   GP1:
	UF : 0, UT : 6,		CONFIG : 'N U T, 0, 0, 0',
	X =  -13.903  mm,	Y =   -293.878  mm,	Z =   -262.975  mm,
	W =  90.000 deg,	P =   0.000 deg,	R =   90.000 deg
};
P[961]{
   GP1:
	UF : 0, UT : 6,		CONFIG : 'N U T, 0, 0, 0',
	X =  -15.345  mm,	Y =   -294.747  mm,	Z =   -263.064  mm,
	W =  90.000 deg,	P =   0.000 deg,	R =   90.000 deg
};
P[962]{
   GP1:
	UF : 0, UT : 6,		CONFIG : 'N U T, 0, 0, 0',
	X =  -16.296  mm,	Y =   -295.198  mm,	Z =   -262.828  mm,
	W =  90.000 deg,	P =   0.000 deg,	R =   90.000 deg
};
P[963]{
   GP1:
	UF : 0, UT : 6,		CONFIG : 'N U T, 0, 0, 0',
	X =  -22.082  mm,	Y =   -298.556  mm,	Z =   -262.870  mm,
	W =  90.000 deg,	P =   0.000 deg,	R =   90.000 deg
};
P[964]{
   GP1:
	UF : 0, UT : 6,		CONFIG : 'N U T, 0, 0, 0',
	X =  -23.322  mm,	Y =   -299.338  mm,	Z =   -263.027  mm,
	W =  90.000 deg,	P =   0.000 deg,	R =   90.000 deg
};
P[965]{
   GP1:
	UF : 0, UT : 6,		CONFIG : 'N U T, 0, 0, 0',
	X =  -24.006  mm,	Y =   -299.749  mm,	Z =   -263.069  mm,
	W =  90.000 deg,	P =   0.000 deg,	R =   90.000 deg
};
P[966]{
   GP1:
	UF : 0, UT : 6,		CONFIG : 'N U T, 0, 0, 0',
	X =  -25.131  mm,	Y =   -300.448  mm,	Z =   -263.189  mm,
	W =  90.000 deg,	P =   0.000 deg,	R =   90.000 deg
};
P[967]{
   GP1:
	UF : 0, UT : 6,		CONFIG : 'N U T, 0, 0, 0',
	X =  -26.021  mm,	Y =   -300.924  mm,	Z =   -263.096  mm,
	W =  90.000 deg,	P =   0.000 deg,	R =   90.000 deg
};
P[968]{
   GP1:
	UF : 0, UT : 6,		CONFIG : 'N U T, 0, 0, 0',
	X =  -27.003  mm,	Y =   -301.481  mm,	Z =   -263.073  mm,
	W =  90.000 deg,	P =   0.000 deg,	R =   90.000 deg
};
P[969]{
   GP1:
	UF : 0, UT : 6,		CONFIG : 'N U T, 0, 0, 0',
	X =  -28.049  mm,	Y =   -302.147  mm,	Z =   -263.222  mm,
	W =  90.000 deg,	P =   0.000 deg,	R =   90.000 deg
};
P[970]{
   GP1:
	UF : 0, UT : 6,		CONFIG : 'N U T, 0, 0, 0',
	X =  -28.885  mm,	Y =   -302.634  mm,	Z =   -263.233  mm,
	W =  90.000 deg,	P =   0.000 deg,	R =   90.000 deg
};
P[971]{
   GP1:
	UF : 0, UT : 6,		CONFIG : 'N U T, 0, 0, 0',
	X =  -30.078  mm,	Y =   -303.309  mm,	Z =   -263.202  mm,
	W =  90.000 deg,	P =   0.000 deg,	R =   90.000 deg
};
P[972]{
   GP1:
	UF : 0, UT : 6,		CONFIG : 'N U T, 0, 0, 0',
	X =  -34.857  mm,	Y =   -305.939  mm,	Z =   -262.886  mm,
	W =  90.000 deg,	P =   0.000 deg,	R =   90.000 deg
};
P[973]{
   GP1:
	UF : 0, UT : 6,		CONFIG : 'N U T, 0, 0, 0',
	X =  -36.596  mm,	Y =   -307.068  mm,	Z =   -263.190  mm,
	W =  90.000 deg,	P =   0.000 deg,	R =   90.000 deg
};
P[974]{
   GP1:
	UF : 0, UT : 6,		CONFIG : 'N U T, 0, 0, 0',
	X =  -40.566  mm,	Y =   -309.197  mm,	Z =   -262.792  mm,
	W =  90.000 deg,	P =   0.000 deg,	R =   90.000 deg
};
P[975]{
   GP1:
	UF : 0, UT : 6,		CONFIG : 'N U T, 0, 0, 0',
	X =  -41.702  mm,	Y =   -309.999  mm,	Z =   -263.147  mm,
	W =  90.000 deg,	P =   0.000 deg,	R =   90.000 deg
};
P[976]{
   GP1:
	UF : 0, UT : 6,		CONFIG : 'N U T, 0, 0, 0',
	X =  -43.375  mm,	Y =   -310.890  mm,	Z =   -262.965  mm,
	W =  90.000 deg,	P =   0.000 deg,	R =   90.000 deg
};
P[977]{
   GP1:
	UF : 0, UT : 6,		CONFIG : 'N U T, 0, 0, 0',
	X =  -45.750  mm,	Y =   -312.335  mm,	Z =   -263.145  mm,
	W =  90.000 deg,	P =   0.000 deg,	R =   90.000 deg
};
P[978]{
   GP1:
	UF : 0, UT : 6,		CONFIG : 'N U T, 0, 0, 0',
	X =  -46.386  mm,	Y =   -312.642  mm,	Z =   -262.998  mm,
	W =  90.000 deg,	P =   0.000 deg,	R =   90.000 deg
};
P[979]{
   GP1:
	UF : 0, UT : 6,		CONFIG : 'N U T, 0, 0, 0',
	X =  -48.196  mm,	Y =   -313.624  mm,	Z =   -262.843  mm,
	W =  90.000 deg,	P =   0.000 deg,	R =   90.000 deg
};
P[980]{
   GP1:
	UF : 0, UT : 6,		CONFIG : 'N U T, 0, 0, 0',
	X =  -49.126  mm,	Y =   -314.230  mm,	Z =   -263.010  mm,
	W =  90.000 deg,	P =   0.000 deg,	R =   90.000 deg
};
P[981]{
   GP1:
	UF : 0, UT : 6,		CONFIG : 'N U T, 0, 0, 0',
	X =  -50.042  mm,	Y =   -314.775  mm,	Z =   -263.050  mm,
	W =  90.000 deg,	P =   0.000 deg,	R =   90.000 deg
};
P[982]{
   GP1:
	UF : 0, UT : 6,		CONFIG : 'N U T, 0, 0, 0',
	X =  -53.055  mm,	Y =   -316.565  mm,	Z =   -263.174  mm,
	W =  90.000 deg,	P =   0.000 deg,	R =   90.000 deg
};
P[983]{
   GP1:
	UF : 0, UT : 6,		CONFIG : 'N U T, 0, 0, 0',
	X =  -55.480  mm,	Y =   -317.838  mm,	Z =   -262.864  mm,
	W =  90.000 deg,	P =   0.000 deg,	R =   90.000 deg
};
P[984]{
   GP1:
	UF : 0, UT : 6,		CONFIG : 'N U T, 0, 0, 0',
	X =  -57.242  mm,	Y =   -318.967  mm,	Z =   -263.135  mm,
	W =  90.000 deg,	P =   0.000 deg,	R =   90.000 deg
};
P[985]{
   GP1:
	UF : 0, UT : 6,		CONFIG : 'N U T, 0, 0, 0',
	X =  -58.253  mm,	Y =   -319.525  mm,	Z =   -263.074  mm,
	W =  90.000 deg,	P =   0.000 deg,	R =   90.000 deg
};
P[986]{
   GP1:
	UF : 0, UT : 6,		CONFIG : 'N U T, 0, 0, 0',
	X =  -59.249  mm,	Y =   -320.111  mm,	Z =   -263.099  mm,
	W =  90.000 deg,	P =   0.000 deg,	R =   90.000 deg
};
P[987]{
   GP1:
	UF : 0, UT : 6,		CONFIG : 'N U T, 0, 0, 0',
	X =  -60.340  mm,	Y =   -320.605  mm,	Z =   -262.770  mm,
	W =  90.000 deg,	P =   0.000 deg,	R =   90.000 deg
};
P[988]{
   GP1:
	UF : 0, UT : 6,		CONFIG : 'N U T, 0, 0, 0',
	X =  -62.108  mm,	Y =   -321.686  mm,	Z =   -262.916  mm,
	W =  90.000 deg,	P =   0.000 deg,	R =   90.000 deg
};
P[989]{
   GP1:
	UF : 0, UT : 6,		CONFIG : 'N U T, 0, 0, 0',
	X =  -62.787  mm,	Y =   -322.064  mm,	Z =   -262.884  mm,
	W =  90.000 deg,	P =   0.000 deg,	R =   90.000 deg
};
P[990]{
   GP1:
	UF : 0, UT : 6,		CONFIG : 'N U T, 0, 0, 0',
	X =  -64.134  mm,	Y =   -322.855  mm,	Z =   -262.913  mm,
	W =  90.000 deg,	P =   0.000 deg,	R =   90.000 deg
};
P[991]{
   GP1:
	UF : 0, UT : 6,		CONFIG : 'N U T, 0, 0, 0',
	X =  -66.215  mm,	Y =   -324.115  mm,	Z =   -263.054  mm,
	W =  90.000 deg,	P =   0.000 deg,	R =   90.000 deg
};
P[992]{
   GP1:
	UF : 0, UT : 6,		CONFIG : 'N U T, 0, 0, 0',
	X =  -67.562  mm,	Y =   -324.948  mm,	Z =   -263.191  mm,
	W =  90.000 deg,	P =   0.000 deg,	R =   90.000 deg
};
P[993]{
   GP1:
	UF : 0, UT : 6,		CONFIG : 'N U T, 0, 0, 0',
	X =  -69.553  mm,	Y =   -326.046  mm,	Z =   -263.064  mm,
	W =  90.000 deg,	P =   0.000 deg,	R =   90.000 deg
};
P[994]{
   GP1:
	UF : 0, UT : 6,		CONFIG : 'N U T, 0, 0, 0',
	X =  -70.474  mm,	Y =   -326.519  mm,	Z =   -262.920  mm,
	W =  90.000 deg,	P =   0.000 deg,	R =   90.000 deg
};
P[995]{
   GP1:
	UF : 0, UT : 6,		CONFIG : 'N U T, 0, 0, 0',
	X =  -71.598  mm,	Y =   -327.225  mm,	Z =   -263.060  mm,
	W =  90.000 deg,	P =   0.000 deg,	R =   90.000 deg
};
P[996]{
   GP1:
	UF : 0, UT : 6,		CONFIG : 'N U T, 0, 0, 0',
	X =  -74.940  mm,	Y =   -329.214  mm,	Z =   -263.203  mm,
	W =  90.000 deg,	P =   0.000 deg,	R =   90.000 deg
};
P[997]{
   GP1:
	UF : 0, UT : 6,		CONFIG : 'N U T, 0, 0, 0',
	X =  -75.933  mm,	Y =   -329.603  mm,	Z =   -262.758  mm,
	W =  90.000 deg,	P =   0.000 deg,	R =   90.000 deg
};
P[998]{
   GP1:
	UF : 0, UT : 6,		CONFIG : 'N U T, 0, 0, 0',
	X =  -76.875  mm,	Y =   -330.326  mm,	Z =   -263.193  mm,
	W =  90.000 deg,	P =   0.000 deg,	R =   90.000 deg
};
P[999]{
   GP1:
	UF : 0, UT : 6,		CONFIG : 'N U T, 0, 0, 0',
	X =  -79.257  mm,	Y =   -331.581  mm,	Z =   -262.899  mm,
	W =  90.000 deg,	P =   0.000 deg,	R =   90.000 deg
};
P[1000]{
   GP1:
	UF : 0, UT : 6,		CONFIG : 'N U T, 0, 0, 0',
	X =  -80.224  mm,	Y =   -332.210  mm,	Z =   -263.072  mm,
	W =  90.000 deg,	P =   0.000 deg,	R =   90.000 deg
};
P[1001]{
   GP1:
	UF : 0, UT : 6,		CONFIG : 'N U T, 0, 0, 0',
	X =  -81.301  mm,	Y =   -332.796  mm,	Z =   -262.984  mm,
	W =  90.000 deg,	P =   0.000 deg,	R =   90.000 deg
};
P[1002]{
   GP1:
	UF : 0, UT : 6,		CONFIG : 'N U T, 0, 0, 0',
	X =  -82.537  mm,	Y =   -333.595  mm,	Z =   -263.191  mm,
	W =  90.000 deg,	P =   0.000 deg,	R =   90.000 deg
};
P[1003]{
   GP1:
	UF : 0, UT : 6,		CONFIG : 'N U T, 0, 0, 0',
	X =  -84.221  mm,	Y =   -334.495  mm,	Z =   -263.013  mm,
	W =  90.000 deg,	P =   0.000 deg,	R =   90.000 deg
};
P[1004]{
   GP1:
	UF : 0, UT : 6,		CONFIG : 'N U T, 0, 0, 0',
	X =  -86.503  mm,	Y =   -335.901  mm,	Z =   -263.231  mm,
	W =  90.000 deg,	P =   0.000 deg,	R =   90.000 deg
};
P[1005]{
   GP1:
	UF : 0, UT : 6,		CONFIG : 'N U T, 0, 0, 0',
	X =  -87.830  mm,	Y =   -336.582  mm,	Z =   -263.024  mm,
	W =  90.000 deg,	P =   0.000 deg,	R =   90.000 deg
};
P[1006]{
   GP1:
	UF : 0, UT : 6,		CONFIG : 'N U T, 0, 0, 0',
	X =  -88.563  mm,	Y =   -336.971  mm,	Z =   -262.940  mm,
	W =  90.000 deg,	P =   0.000 deg,	R =   90.000 deg
};
P[1007]{
   GP1:
	UF : 0, UT : 6,		CONFIG : 'N U T, 0, 0, 0',
	X =  -91.169  mm,	Y =   -338.484  mm,	Z =   -262.960  mm,
	W =  90.000 deg,	P =   0.000 deg,	R =   90.000 deg
};
P[1008]{
   GP1:
	UF : 0, UT : 6,		CONFIG : 'N U T, 0, 0, 0',
	X =  -91.807  mm,	Y =   -338.966  mm,	Z =   -263.237  mm,
	W =  90.000 deg,	P =   0.000 deg,	R =   90.000 deg
};
P[1009]{
   GP1:
	UF : 0, UT : 6,		CONFIG : 'N U T, 0, 0, 0',
	X =  -92.493  mm,	Y =   -339.305  mm,	Z =   -263.100  mm,
	W =  90.000 deg,	P =   0.000 deg,	R =   90.000 deg
};
P[1010]{
   GP1:
	UF : 0, UT : 6,		CONFIG : 'N U T, 0, 0, 0',
	X =  -93.733  mm,	Y =   -340.067  mm,	Z =   -263.210  mm,
	W =  90.000 deg,	P =   0.000 deg,	R =   90.000 deg
};
P[1011]{
   GP1:
	UF : 0, UT : 6,		CONFIG : 'N U T, 0, 0, 0',
	X =  -95.528  mm,	Y =   -341.015  mm,	Z =   -262.997  mm,
	W =  90.000 deg,	P =   0.000 deg,	R =   90.000 deg
};
P[1012]{
   GP1:
	UF : 0, UT : 6,		CONFIG : 'N U T, 0, 0, 0',
	X =  -96.099  mm,	Y =   -341.423  mm,	Z =   -263.185  mm,
	W =  90.000 deg,	P =   0.000 deg,	R =   90.000 deg
};
P[1013]{
   GP1:
	UF : 0, UT : 6,		CONFIG : 'N U T, 0, 0, 0',
	X =  -97.870  mm,	Y =   -342.351  mm,	Z =   -262.957  mm,
	W =  90.000 deg,	P =   0.000 deg,	R =   90.000 deg
};
P[1014]{
   GP1:
	UF : 0, UT : 6,		CONFIG : 'N U T, 0, 0, 0',
	X =  -98.558  mm,	Y =   -342.684  mm,	Z =   -262.799  mm,
	W =  90.000 deg,	P =   0.000 deg,	R =   90.000 deg
};
P[1015]{
   GP1:
	UF : 0, UT : 6,		CONFIG : 'N U T, 0, 0, 0',
	X =  -100.265  mm,	Y =   -343.664  mm,	Z =   -262.786  mm,
	W =  90.000 deg,	P =   0.000 deg,	R =   90.000 deg
};
P[1016]{
   GP1:
	UF : 0, UT : 6,		CONFIG : 'N U T, 0, 0, 0',
	X =  -101.104  mm,	Y =   -344.315  mm,	Z =   -263.189  mm,
	W =  90.000 deg,	P =   0.000 deg,	R =   90.000 deg
};
P[1017]{
   GP1:
	UF : 0, UT : 6,		CONFIG : 'N U T, 0, 0, 0',
	X =  -102.677  mm,	Y =   -345.092  mm,	Z =   -262.871  mm,
	W =  90.000 deg,	P =   0.000 deg,	R =   90.000 deg
};
P[1018]{
   GP1:
	UF : 0, UT : 6,		CONFIG : 'N U T, 0, 0, 0',
	X =  -103.616  mm,	Y =   -345.734  mm,	Z =   -263.113  mm,
	W =  90.000 deg,	P =   0.000 deg,	R =   90.000 deg
};
P[1019]{
   GP1:
	UF : 0, UT : 6,		CONFIG : 'N U T, 0, 0, 0',
	X =  -107.113  mm,	Y =   -347.775  mm,	Z =   -263.168  mm,
	W =  90.000 deg,	P =   0.000 deg,	R =   90.000 deg
};
P[1020]{
   GP1:
	UF : 0, UT : 6,		CONFIG : 'N U T, 0, 0, 0',
	X =  -109.559  mm,	Y =   -349.127  mm,	Z =   -263.019  mm,
	W =  90.000 deg,	P =   0.000 deg,	R =   90.000 deg
};
P[1021]{
   GP1:
	UF : 0, UT : 6,		CONFIG : 'N U T, 0, 0, 0',
	X =  -110.422  mm,	Y =   -349.715  mm,	Z =   -263.238  mm,
	W =  90.000 deg,	P =   0.000 deg,	R =   90.000 deg
};
P[1022]{
   GP1:
	UF : 0, UT : 6,		CONFIG : 'N U T, 0, 0, 0',
	X =  -111.709  mm,	Y =   -350.433  mm,	Z =   -263.142  mm,
	W =  90.000 deg,	P =   0.000 deg,	R =   90.000 deg
};
P[1023]{
   GP1:
	UF : 0, UT : 6,		CONFIG : 'N U T, 0, 0, 0',
	X =  -114.563  mm,	Y =   -352.669  mm,	Z =   -263.167  mm,
	W =  90.000 deg,	P =   0.000 deg,	R =   90.000 deg
};
P[1024]{
   GP1:
	UF : 0, UT : 6,		CONFIG : 'N U T, 0, 0, 0',
	X =  -115.198  mm,	Y =   -353.316  mm,	Z =   -263.069  mm,
	W =  90.000 deg,	P =   0.000 deg,	R =   90.000 deg
};
P[1025]{
   GP1:
	UF : 0, UT : 6,		CONFIG : 'N U T, 0, 0, 0',
	X =  -117.423  mm,	Y =   -356.705  mm,	Z =   -263.118  mm,
	W =  90.000 deg,	P =   0.000 deg,	R =   90.000 deg
};
P[1026]{
   GP1:
	UF : 0, UT : 6,		CONFIG : 'N U T, 0, 0, 0',
	X =  -117.726  mm,	Y =   -357.586  mm,	Z =   -263.245  mm,
	W =  90.000 deg,	P =   0.000 deg,	R =   90.000 deg
};
P[1027]{
   GP1:
	UF : 0, UT : 6,		CONFIG : 'N U T, 0, 0, 0',
	X =  -118.115  mm,	Y =   -358.723  mm,	Z =   -263.116  mm,
	W =  90.000 deg,	P =   0.000 deg,	R =   90.000 deg
};
P[1028]{
   GP1:
	UF : 0, UT : 6,		CONFIG : 'N U T, 0, 0, 0',
	X =  -118.602  mm,	Y =   -361.256  mm,	Z =   -262.992  mm,
	W =  90.000 deg,	P =   0.000 deg,	R =   90.000 deg
};
P[1029]{
   GP1:
	UF : 0, UT : 6,		CONFIG : 'N U T, 0, 0, 0',
	X =  -118.574  mm,	Y =   -363.321  mm,	Z =   -263.077  mm,
	W =  90.000 deg,	P =   0.000 deg,	R =   90.000 deg
};
P[1030]{
   GP1:
	UF : 0, UT : 6,		CONFIG : 'N U T, 0, 0, 0',
	X =  -118.207  mm,	Y =   -365.061  mm,	Z =   -263.179  mm,
	W =  90.000 deg,	P =   0.000 deg,	R =   90.000 deg
};
P[1031]{
   GP1:
	UF : 0, UT : 6,		CONFIG : 'N U T, 0, 0, 0',
	X =  -117.889  mm,	Y =   -366.383  mm,	Z =   -263.224  mm,
	W =  90.000 deg,	P =   0.000 deg,	R =   90.000 deg
};
P[1032]{
   GP1:
	UF : 0, UT : 6,		CONFIG : 'N U T, 0, 0, 0',
	X =  -117.012  mm,	Y =   -368.554  mm,	Z =   -263.053  mm,
	W =  90.000 deg,	P =   0.000 deg,	R =   90.000 deg
};
P[1033]{
   GP1:
	UF : 0, UT : 6,		CONFIG : 'N U T, 0, 0, 0',
	X =  -116.322  mm,	Y =   -369.824  mm,	Z =   -263.139  mm,
	W =  90.000 deg,	P =   0.000 deg,	R =   90.000 deg
};
P[1034]{
   GP1:
	UF : 0, UT : 6,		CONFIG : 'N U T, 0, 0, 0',
	X =  -115.983  mm,	Y =   -370.432  mm,	Z =   -263.111  mm,
	W =  90.000 deg,	P =   0.000 deg,	R =   90.000 deg
};
P[1035]{
   GP1:
	UF : 0, UT : 6,		CONFIG : 'N U T, 0, 0, 0',
	X =  -115.285  mm,	Y =   -371.743  mm,	Z =   -262.966  mm,
	W =  90.000 deg,	P =   0.000 deg,	R =   90.000 deg
};
P[1036]{
   GP1:
	UF : 0, UT : 6,		CONFIG : 'N U T, 0, 0, 0',
	X =  -114.882  mm,	Y =   -372.354  mm,	Z =   -263.089  mm,
	W =  90.000 deg,	P =   0.000 deg,	R =   90.000 deg
};
P[1037]{
   GP1:
	UF : 0, UT : 6,		CONFIG : 'N U T, 0, 0, 0',
	X =  -113.584  mm,	Y =   -374.650  mm,	Z =   -263.021  mm,
	W =  90.000 deg,	P =   0.000 deg,	R =   90.000 deg
};
P[1038]{
   GP1:
	UF : 0, UT : 6,		CONFIG : 'N U T, 0, 0, 0',
	X =  -112.392  mm,	Y =   -376.883  mm,	Z =   -262.787  mm,
	W =  90.000 deg,	P =   0.000 deg,	R =   90.000 deg
};
P[1039]{
   GP1:
	UF : 0, UT : 6,		CONFIG : 'N U T, 0, 0, 0',
	X =  -111.637  mm,	Y =   -377.966  mm,	Z =   -263.099  mm,
	W =  90.000 deg,	P =   0.000 deg,	R =   90.000 deg
};
P[1040]{
   GP1:
	UF : 0, UT : 6,		CONFIG : 'N U T, 0, 0, 0',
	X =  -107.435  mm,	Y =   -385.253  mm,	Z =   -263.085  mm,
	W =  90.000 deg,	P =   0.000 deg,	R =   90.000 deg
};
P[1041]{
   GP1:
	UF : 0, UT : 6,		CONFIG : 'N U T, 0, 0, 0',
	X =  -106.804  mm,	Y =   -386.568  mm,	Z =   -262.775  mm,
	W =  90.000 deg,	P =   0.000 deg,	R =   90.000 deg
};
P[1042]{
   GP1:
	UF : 0, UT : 6,		CONFIG : 'N U T, 0, 0, 0',
	X =  -105.774  mm,	Y =   -388.206  mm,	Z =   -262.982  mm,
	W =  90.000 deg,	P =   0.000 deg,	R =   90.000 deg
};
P[1043]{
   GP1:
	UF : 0, UT : 6,		CONFIG : 'N U T, 0, 0, 0',
	X =  -105.097  mm,	Y =   -389.195  mm,	Z =   -263.237  mm,
	W =  90.000 deg,	P =   0.000 deg,	R =   90.000 deg
};
P[1044]{
   GP1:
	UF : 0, UT : 6,		CONFIG : 'N U T, 0, 0, 0',
	X =  -104.414  mm,	Y =   -390.491  mm,	Z =   -263.078  mm,
	W =  90.000 deg,	P =   0.000 deg,	R =   90.000 deg
};
P[1045]{
   GP1:
	UF : 0, UT : 6,		CONFIG : 'N U T, 0, 0, 0',
	X =  -103.894  mm,	Y =   -391.411  mm,	Z =   -263.052  mm,
	W =  90.000 deg,	P =   0.000 deg,	R =   90.000 deg
};
P[1046]{
   GP1:
	UF : 0, UT : 6,		CONFIG : 'N U T, 0, 0, 0',
	X =  -103.256  mm,	Y =   -392.421  mm,	Z =   -263.184  mm,
	W =  90.000 deg,	P =   0.000 deg,	R =   90.000 deg
};
P[1047]{
   GP1:
	UF : 0, UT : 6,		CONFIG : 'N U T, 0, 0, 0',
	X =  -102.760  mm,	Y =   -393.344  mm,	Z =   -263.095  mm,
	W =  90.000 deg,	P =   0.000 deg,	R =   90.000 deg
};
P[1048]{
   GP1:
	UF : 0, UT : 6,		CONFIG : 'N U T, 0, 0, 0',
	X =  -101.499  mm,	Y =   -395.746  mm,	Z =   -262.790  mm,
	W =  90.000 deg,	P =   0.000 deg,	R =   90.000 deg
};
P[1049]{
   GP1:
	UF : 0, UT : 6,		CONFIG : 'N U T, 0, 0, 0',
	X =  -100.798  mm,	Y =   -396.817  mm,	Z =   -262.989  mm,
	W =  90.000 deg,	P =   0.000 deg,	R =   90.000 deg
};
P[1050]{
   GP1:
	UF : 0, UT : 6,		CONFIG : 'N U T, 0, 0, 0',
	X =  -99.795  mm,	Y =   -398.512  mm,	Z =   -263.050  mm,
	W =  90.000 deg,	P =   0.000 deg,	R =   90.000 deg
};
P[1051]{
   GP1:
	UF : 0, UT : 6,		CONFIG : 'N U T, 0, 0, 0',
	X =  -99.179  mm,	Y =   -399.555  mm,	Z =   -263.082  mm,
	W =  90.000 deg,	P =   0.000 deg,	R =   90.000 deg
};
P[1052]{
   GP1:
	UF : 0, UT : 6,		CONFIG : 'N U T, 0, 0, 0',
	X =  -97.942  mm,	Y =   -401.662  mm,	Z =   -263.134  mm,
	W =  90.000 deg,	P =   0.000 deg,	R =   90.000 deg
};
P[1053]{
   GP1:
	UF : 0, UT : 6,		CONFIG : 'N U T, 0, 0, 0',
	X =  -97.334  mm,	Y =   -402.964  mm,	Z =   -262.783  mm,
	W =  90.000 deg,	P =   0.000 deg,	R =   90.000 deg
};
P[1054]{
   GP1:
	UF : 0, UT : 6,		CONFIG : 'N U T, 0, 0, 0',
	X =  -96.595  mm,	Y =   -404.228  mm,	Z =   -262.806  mm,
	W =  90.000 deg,	P =   0.000 deg,	R =   90.000 deg
};
P[1055]{
   GP1:
	UF : 0, UT : 6,		CONFIG : 'N U T, 0, 0, 0',
	X =  -95.365  mm,	Y =   -406.151  mm,	Z =   -263.096  mm,
	W =  90.000 deg,	P =   0.000 deg,	R =   90.000 deg
};
P[1056]{
   GP1:
	UF : 0, UT : 6,		CONFIG : 'N U T, 0, 0, 0',
	X =  -94.824  mm,	Y =   -407.301  mm,	Z =   -262.797  mm,
	W =  90.000 deg,	P =   0.000 deg,	R =   90.000 deg
};
P[1057]{
   GP1:
	UF : 0, UT : 6,		CONFIG : 'N U T, 0, 0, 0',
	X =  -93.955  mm,	Y =   -408.499  mm,	Z =   -263.227  mm,
	W =  90.000 deg,	P =   0.000 deg,	R =   90.000 deg
};
P[1058]{
   GP1:
	UF : 0, UT : 6,		CONFIG : 'N U T, 0, 0, 0',
	X =  -93.580  mm,	Y =   -409.387  mm,	Z =   -262.895  mm,
	W =  90.000 deg,	P =   0.000 deg,	R =   90.000 deg
};
P[1059]{
   GP1:
	UF : 0, UT : 6,		CONFIG : 'N U T, 0, 0, 0',
	X =  -92.695  mm,	Y =   -410.733  mm,	Z =   -263.155  mm,
	W =  90.000 deg,	P =   0.000 deg,	R =   90.000 deg
};
P[1060]{
   GP1:
	UF : 0, UT : 6,		CONFIG : 'N U T, 0, 0, 0',
	X =  -90.502  mm,	Y =   -414.497  mm,	Z =   -263.203  mm,
	W =  90.000 deg,	P =   0.000 deg,	R =   90.000 deg
};
P[1061]{
   GP1:
	UF : 0, UT : 6,		CONFIG : 'N U T, 0, 0, 0',
	X =  -89.845  mm,	Y =   -415.741  mm,	Z =   -263.054  mm,
	W =  90.000 deg,	P =   0.000 deg,	R =   90.000 deg
};
P[1062]{
   GP1:
	UF : 0, UT : 6,		CONFIG : 'N U T, 0, 0, 0',
	X =  -89.462  mm,	Y =   -416.470  mm,	Z =   -262.962  mm,
	W =  90.000 deg,	P =   0.000 deg,	R =   90.000 deg
};
P[1063]{
   GP1:
	UF : 0, UT : 6,		CONFIG : 'N U T, 0, 0, 0',
	X =  -89.089  mm,	Y =   -417.185  mm,	Z =   -262.868  mm,
	W =  90.000 deg,	P =   0.000 deg,	R =   90.000 deg
};
P[1064]{
   GP1:
	UF : 0, UT : 6,		CONFIG : 'N U T, 0, 0, 0',
	X =  -87.684  mm,	Y =   -419.644  mm,	Z =   -262.831  mm,
	W =  90.000 deg,	P =   0.000 deg,	R =   90.000 deg
};
P[1065]{
   GP1:
	UF : 0, UT : 6,		CONFIG : 'N U T, 0, 0, 0',
	X =  -87.091  mm,	Y =   -420.612  mm,	Z =   -262.912  mm,
	W =  90.000 deg,	P =   0.000 deg,	R =   90.000 deg
};
P[1066]{
   GP1:
	UF : 0, UT : 6,		CONFIG : 'N U T, 0, 0, 0',
	X =  -86.461  mm,	Y =   -421.515  mm,	Z =   -263.175  mm,
	W =  90.000 deg,	P =   0.000 deg,	R =   90.000 deg
};
P[1067]{
   GP1:
	UF : 0, UT : 6,		CONFIG : 'N U T, 0, 0, 0',
	X =  -85.753  mm,	Y =   -422.744  mm,	Z =   -263.173  mm,
	W =  90.000 deg,	P =   0.000 deg,	R =   90.000 deg
};
P[1068]{
   GP1:
	UF : 0, UT : 6,		CONFIG : 'N U T, 0, 0, 0',
	X =  -84.853  mm,	Y =   -424.493  mm,	Z =   -262.904  mm,
	W =  90.000 deg,	P =   0.000 deg,	R =   90.000 deg
};
P[1069]{
   GP1:
	UF : 0, UT : 6,		CONFIG : 'N U T, 0, 0, 0',
	X =  -82.147  mm,	Y =   -428.978  mm,	Z =   -263.189  mm,
	W =  90.000 deg,	P =   0.000 deg,	R =   90.000 deg
};
P[1070]{
   GP1:
	UF : 0, UT : 6,		CONFIG : 'N U T, 0, 0, 0',
	X =  -81.488  mm,	Y =   -430.368  mm,	Z =   -262.838  mm,
	W =  90.000 deg,	P =   0.000 deg,	R =   90.000 deg
};
P[1071]{
   GP1:
	UF : 0, UT : 6,		CONFIG : 'N U T, 0, 0, 0',
	X =  -80.821  mm,	Y =   -431.485  mm,	Z =   -262.895  mm,
	W =  90.000 deg,	P =   0.000 deg,	R =   90.000 deg
};
P[1072]{
   GP1:
	UF : 0, UT : 6,		CONFIG : 'N U T, 0, 0, 0',
	X =  -80.262  mm,	Y =   -432.225  mm,	Z =   -263.213  mm,
	W =  90.000 deg,	P =   0.000 deg,	R =   90.000 deg
};
P[1073]{
   GP1:
	UF : 0, UT : 6,		CONFIG : 'N U T, 0, 0, 0',
	X =  -78.623  mm,	Y =   -435.273  mm,	Z =   -262.917  mm,
	W =  90.000 deg,	P =   0.000 deg,	R =   90.000 deg
};
P[1074]{
   GP1:
	UF : 0, UT : 6,		CONFIG : 'N U T, 0, 0, 0',
	X =  -77.822  mm,	Y =   -436.615  mm,	Z =   -262.983  mm,
	W =  90.000 deg,	P =   0.000 deg,	R =   90.000 deg
};
P[1075]{
   GP1:
	UF : 0, UT : 6,		CONFIG : 'N U T, 0, 0, 0',
	X =  -77.155  mm,	Y =   -437.636  mm,	Z =   -263.172  mm,
	W =  90.000 deg,	P =   0.000 deg,	R =   90.000 deg
};
P[1076]{
   GP1:
	UF : 0, UT : 6,		CONFIG : 'N U T, 0, 0, 0',
	X =  -76.150  mm,	Y =   -439.438  mm,	Z =   -263.086  mm,
	W =  90.000 deg,	P =   0.000 deg,	R =   90.000 deg
};
P[1077]{
   GP1:
	UF : 0, UT : 6,		CONFIG : 'N U T, 0, 0, 0',
	X =  -75.497  mm,	Y =   -440.686  mm,	Z =   -262.922  mm,
	W =  90.000 deg,	P =   0.000 deg,	R =   90.000 deg
};
P[1078]{
   GP1:
	UF : 0, UT : 6,		CONFIG : 'N U T, 0, 0, 0',
	X =  -73.747  mm,	Y =   -443.722  mm,	Z =   -262.912  mm,
	W =  90.000 deg,	P =   0.000 deg,	R =   90.000 deg
};
P[1079]{
   GP1:
	UF : 0, UT : 6,		CONFIG : 'N U T, 0, 0, 0',
	X =  -73.249  mm,	Y =   -444.554  mm,	Z =   -262.957  mm,
	W =  90.000 deg,	P =   0.000 deg,	R =   90.000 deg
};
P[1080]{
   GP1:
	UF : 0, UT : 6,		CONFIG : 'N U T, 0, 0, 0',
	X =  -72.020  mm,	Y =   -446.678  mm,	Z =   -262.963  mm,
	W =  90.000 deg,	P =   0.000 deg,	R =   90.000 deg
};
P[1081]{
   GP1:
	UF : 0, UT : 6,		CONFIG : 'N U T, 0, 0, 0',
	X =  -71.491  mm,	Y =   -447.557  mm,	Z =   -263.017  mm,
	W =  90.000 deg,	P =   0.000 deg,	R =   90.000 deg
};
P[1082]{
   GP1:
	UF : 0, UT : 6,		CONFIG : 'N U T, 0, 0, 0',
	X =  -68.260  mm,	Y =   -453.237  mm,	Z =   -262.897  mm,
	W =  90.000 deg,	P =   0.000 deg,	R =   90.000 deg
};
P[1083]{
   GP1:
	UF : 0, UT : 6,		CONFIG : 'N U T, 0, 0, 0',
	X =  -66.554  mm,	Y =   -456.053  mm,	Z =   -263.092  mm,
	W =  90.000 deg,	P =   0.000 deg,	R =   90.000 deg
};
P[1084]{
   GP1:
	UF : 0, UT : 6,		CONFIG : 'N U T, 0, 0, 0',
	X =  -64.066  mm,	Y =   -460.264  mm,	Z =   -263.227  mm,
	W =  90.000 deg,	P =   0.000 deg,	R =   90.000 deg
};
P[1085]{
   GP1:
	UF : 0, UT : 6,		CONFIG : 'N U T, 0, 0, 0',
	X =  -63.745  mm,	Y =   -461.131  mm,	Z =   -262.793  mm,
	W =  90.000 deg,	P =   0.000 deg,	R =   90.000 deg
};
P[1086]{
   GP1:
	UF : 0, UT : 6,		CONFIG : 'N U T, 0, 0, 0',
	X =  -61.359  mm,	Y =   -464.951  mm,	Z =   -263.231  mm,
	W =  90.000 deg,	P =   0.000 deg,	R =   90.000 deg
};
P[1087]{
   GP1:
	UF : 0, UT : 6,		CONFIG : 'N U T, 0, 0, 0',
	X =  -60.085  mm,	Y =   -467.217  mm,	Z =   -263.147  mm,
	W =  90.000 deg,	P =   0.000 deg,	R =   90.000 deg
};
P[1088]{
   GP1:
	UF : 0, UT : 6,		CONFIG : 'N U T, 0, 0, 0',
	X =  -59.296  mm,	Y =   -468.735  mm,	Z =   -262.934  mm,
	W =  90.000 deg,	P =   0.000 deg,	R =   90.000 deg
};
P[1089]{
   GP1:
	UF : 0, UT : 6,		CONFIG : 'N U T, 0, 0, 0',
	X =  -58.716  mm,	Y =   -469.717  mm,	Z =   -262.965  mm,
	W =  90.000 deg,	P =   0.000 deg,	R =   90.000 deg
};
P[1090]{
   GP1:
	UF : 0, UT : 6,		CONFIG : 'N U T, 0, 0, 0',
	X =  -58.101  mm,	Y =   -470.743  mm,	Z =   -263.019  mm,
	W =  90.000 deg,	P =   0.000 deg,	R =   90.000 deg
};
P[1091]{
   GP1:
	UF : 0, UT : 6,		CONFIG : 'N U T, 0, 0, 0',
	X =  -57.668  mm,	Y =   -471.616  mm,	Z =   -262.847  mm,
	W =  90.000 deg,	P =   0.000 deg,	R =   90.000 deg
};
P[1092]{
   GP1:
	UF : 0, UT : 6,		CONFIG : 'N U T, 0, 0, 0',
	X =  -56.102  mm,	Y =   -474.080  mm,	Z =   -263.194  mm,
	W =  90.000 deg,	P =   0.000 deg,	R =   90.000 deg
};
P[1093]{
   GP1:
	UF : 0, UT : 6,		CONFIG : 'N U T, 0, 0, 0',
	X =  -54.772  mm,	Y =   -476.607  mm,	Z =   -262.882  mm,
	W =  90.000 deg,	P =   0.000 deg,	R =   90.000 deg
};
P[1094]{
   GP1:
	UF : 0, UT : 6,		CONFIG : 'N U T, 0, 0, 0',
	X =  -53.834  mm,	Y =   -478.104  mm,	Z =   -263.060  mm,
	W =  90.000 deg,	P =   0.000 deg,	R =   90.000 deg
};
P[1095]{
   GP1:
	UF : 0, UT : 6,		CONFIG : 'N U T, 0, 0, 0',
	X =  -53.421  mm,	Y =   -478.798  mm,	Z =   -263.091  mm,
	W =  90.000 deg,	P =   0.000 deg,	R =   90.000 deg
};
P[1096]{
   GP1:
	UF : 0, UT : 6,		CONFIG : 'N U T, 0, 0, 0',
	X =  -52.867  mm,	Y =   -479.903  mm,	Z =   -262.889  mm,
	W =  90.000 deg,	P =   0.000 deg,	R =   90.000 deg
};
P[1097]{
   GP1:
	UF : 0, UT : 6,		CONFIG : 'N U T, 0, 0, 0',
	X =  -52.447  mm,	Y =   -480.576  mm,	Z =   -262.964  mm,
	W =  90.000 deg,	P =   0.000 deg,	R =   90.000 deg
};
P[1098]{
   GP1:
	UF : 0, UT : 6,		CONFIG : 'N U T, 0, 0, 0',
	X =  -50.365  mm,	Y =   -484.077  mm,	Z =   -263.110  mm,
	W =  90.000 deg,	P =   0.000 deg,	R =   90.000 deg
};
P[1099]{
   GP1:
	UF : 0, UT : 6,		CONFIG : 'N U T, 0, 0, 0',
	X =  -49.641  mm,	Y =   -485.439  mm,	Z =   -262.960  mm,
	W =  90.000 deg,	P =   0.000 deg,	R =   90.000 deg
};
P[1100]{
   GP1:
	UF : 0, UT : 6,		CONFIG : 'N U T, 0, 0, 0',
	X =  -48.019  mm,	Y =   -488.252  mm,	Z =   -262.954  mm,
	W =  90.000 deg,	P =   0.000 deg,	R =   90.000 deg
};
P[1101]{
   GP1:
	UF : 0, UT : 6,		CONFIG : 'N U T, 0, 0, 0',
	X =  -46.572  mm,	Y =   -490.772  mm,	Z =   -262.935  mm,
	W =  90.000 deg,	P =   0.000 deg,	R =   90.000 deg
};
P[1102]{
   GP1:
	UF : 0, UT : 6,		CONFIG : 'N U T, 0, 0, 0',
	X =  -42.398  mm,	Y =   -497.795  mm,	Z =   -263.222  mm,
	W =  90.000 deg,	P =   0.000 deg,	R =   90.000 deg
};
P[1103]{
   GP1:
	UF : 0, UT : 6,		CONFIG : 'N U T, 0, 0, 0',
	X =  -41.956  mm,	Y =   -498.648  mm,	Z =   -263.101  mm,
	W =  90.000 deg,	P =   0.000 deg,	R =   90.000 deg
};
P[1104]{
   GP1:
	UF : 0, UT : 6,		CONFIG : 'N U T, 0, 0, 0',
	X =  -38.366  mm,	Y =   -504.846  mm,	Z =   -263.130  mm,
	W =  90.000 deg,	P =   0.000 deg,	R =   90.000 deg
};
P[1105]{
   GP1:
	UF : 0, UT : 6,		CONFIG : 'N U T, 0, 0, 0',
	X =  -37.923  mm,	Y =   -505.786  mm,	Z =   -262.884  mm,
	W =  90.000 deg,	P =   0.000 deg,	R =   90.000 deg
};
P[1106]{
   GP1:
	UF : 0, UT : 6,		CONFIG : 'N U T, 0, 0, 0',
	X =  -37.193  mm,	Y =   -507.081  mm,	Z =   -262.845  mm,
	W =  90.000 deg,	P =   0.000 deg,	R =   90.000 deg
};
P[1107]{
   GP1:
	UF : 0, UT : 6,		CONFIG : 'N U T, 0, 0, 0',
	X =  -35.214  mm,	Y =   -510.475  mm,	Z =   -262.891  mm,
	W =  90.000 deg,	P =   0.000 deg,	R =   90.000 deg
};
P[1108]{
   GP1:
	UF : 0, UT : 6,		CONFIG : 'N U T, 0, 0, 0',
	X =  -34.708  mm,	Y =   -511.190  mm,	Z =   -263.114  mm,
	W =  90.000 deg,	P =   0.000 deg,	R =   90.000 deg
};
P[1109]{
   GP1:
	UF : 0, UT : 6,		CONFIG : 'N U T, 0, 0, 0',
	X =  -34.193  mm,	Y =   -512.125  mm,	Z =   -263.057  mm,
	W =  90.000 deg,	P =   0.000 deg,	R =   90.000 deg
};
P[1110]{
   GP1:
	UF : 0, UT : 6,		CONFIG : 'N U T, 0, 0, 0',
	X =  -33.234  mm,	Y =   -513.642  mm,	Z =   -263.257  mm,
	W =  90.000 deg,	P =   0.000 deg,	R =   90.000 deg
};
P[1111]{
   GP1:
	UF : 0, UT : 6,		CONFIG : 'N U T, 0, 0, 0',
	X =  -32.825  mm,	Y =   -514.680  mm,	Z =   -262.794  mm,
	W =  90.000 deg,	P =   0.000 deg,	R =   90.000 deg
};
P[1112]{
   GP1:
	UF : 0, UT : 6,		CONFIG : 'N U T, 0, 0, 0',
	X =  -31.805  mm,	Y =   -516.289  mm,	Z =   -263.017  mm,
	W =  90.000 deg,	P =   0.000 deg,	R =   90.000 deg
};
P[1113]{
   GP1:
	UF : 0, UT : 6,		CONFIG : 'N U T, 0, 0, 0',
	X =  -31.223  mm,	Y =   -517.271  mm,	Z =   -263.052  mm,
	W =  90.000 deg,	P =   0.000 deg,	R =   90.000 deg
};
P[1114]{
   GP1:
	UF : 0, UT : 6,		CONFIG : 'N U T, 0, 0, 0',
	X =  -29.506  mm,	Y =   -520.413  mm,	Z =   -262.819  mm,
	W =  90.000 deg,	P =   0.000 deg,	R =   90.000 deg
};
P[1115]{
   GP1:
	UF : 0, UT : 6,		CONFIG : 'N U T, 0, 0, 0',
	X =  -28.578  mm,	Y =   -521.840  mm,	Z =   -263.070  mm,
	W =  90.000 deg,	P =   0.000 deg,	R =   90.000 deg
};
P[1116]{
   GP1:
	UF : 0, UT : 6,		CONFIG : 'N U T, 0, 0, 0',
	X =  -27.948  mm,	Y =   -523.034  mm,	Z =   -262.928  mm,
	W =  90.000 deg,	P =   0.000 deg,	R =   90.000 deg
};
P[1117]{
   GP1:
	UF : 0, UT : 6,		CONFIG : 'N U T, 0, 0, 0',
	X =  -27.308  mm,	Y =   -524.005  mm,	Z =   -263.118  mm,
	W =  90.000 deg,	P =   0.000 deg,	R =   90.000 deg
};
P[1118]{
   GP1:
	UF : 0, UT : 6,		CONFIG : 'N U T, 0, 0, 0',
	X =  -26.829  mm,	Y =   -524.923  mm,	Z =   -262.992  mm,
	W =  90.000 deg,	P =   0.000 deg,	R =   90.000 deg
};
P[1119]{
   GP1:
	UF : 0, UT : 6,		CONFIG : 'N U T, 0, 0, 0',
	X =  -25.904  mm,	Y =   -526.498  mm,	Z =   -263.032  mm,
	W =  90.000 deg,	P =   0.000 deg,	R =   90.000 deg
};
P[1120]{
   GP1:
	UF : 0, UT : 6,		CONFIG : 'N U T, 0, 0, 0',
	X =  -24.521  mm,	Y =   -529.018  mm,	Z =   -262.859  mm,
	W =  90.000 deg,	P =   0.000 deg,	R =   90.000 deg
};
P[1121]{
   GP1:
	UF : 0, UT : 6,		CONFIG : 'N U T, 0, 0, 0',
	X =  -24.057  mm,	Y =   -529.604  mm,	Z =   -263.162  mm,
	W =  90.000 deg,	P =   0.000 deg,	R =   90.000 deg
};
P[1122]{
   GP1:
	UF : 0, UT : 6,		CONFIG : 'N U T, 0, 0, 0',
	X =  -23.696  mm,	Y =   -530.396  mm,	Z =   -262.930  mm,
	W =  90.000 deg,	P =   0.000 deg,	R =   90.000 deg
};
P[1123]{
   GP1:
	UF : 0, UT : 6,		CONFIG : 'N U T, 0, 0, 0',
	X =  -22.832  mm,	Y =   -531.741  mm,	Z =   -263.141  mm,
	W =  90.000 deg,	P =   0.000 deg,	R =   90.000 deg
};
P[1124]{
   GP1:
	UF : 0, UT : 6,		CONFIG : 'N U T, 0, 0, 0',
	X =  -17.699  mm,	Y =   -540.894  mm,	Z =   -262.770  mm,
	W =  90.000 deg,	P =   0.000 deg,	R =   90.000 deg
};
P[1125]{
   GP1:
	UF : 0, UT : 6,		CONFIG : 'N U T, 0, 0, 0',
	X =  -16.483  mm,	Y =   -542.930  mm,	Z =   -262.868  mm,
	W =  90.000 deg,	P =   0.000 deg,	R =   90.000 deg
};
P[1126]{
   GP1:
	UF : 0, UT : 6,		CONFIG : 'N U T, 0, 0, 0',
	X =  -16.139  mm,	Y =   -543.605  mm,	Z =   -262.759  mm,
	W =  90.000 deg,	P =   0.000 deg,	R =   90.000 deg
};
P[1127]{
   GP1:
	UF : 0, UT : 6,		CONFIG : 'N U T, 0, 0, 0',
	X =  -15.752  mm,	Y =   -543.956  mm,	Z =   -263.207  mm,
	W =  90.000 deg,	P =   0.000 deg,	R =   90.000 deg
};
P[1128]{
   GP1:
	UF : 0, UT : 6,		CONFIG : 'N U T, 0, 0, 0',
	X =  -15.298  mm,	Y =   -544.876  mm,	Z =   -263.019  mm,
	W =  90.000 deg,	P =   0.000 deg,	R =   90.000 deg
};
P[1129]{
   GP1:
	UF : 0, UT : 6,		CONFIG : 'N U T, 0, 0, 0',
	X =  -14.990  mm,	Y =   -545.575  mm,	Z =   -262.786  mm,
	W =  90.000 deg,	P =   0.000 deg,	R =   90.000 deg
};
P[1130]{
   GP1:
	UF : 0, UT : 6,		CONFIG : 'N U T, 0, 0, 0',
	X =  -14.187  mm,	Y =   -546.930  mm,	Z =   -262.837  mm,
	W =  90.000 deg,	P =   0.000 deg,	R =   90.000 deg
};
P[1131]{
   GP1:
	UF : 0, UT : 6,		CONFIG : 'N U T, 0, 0, 0',
	X =  -13.674  mm,	Y =   -547.529  mm,	Z =   -263.241  mm,
	W =  90.000 deg,	P =   0.000 deg,	R =   90.000 deg
};
P[1132]{
   GP1:
	UF : 0, UT : 6,		CONFIG : 'N U T, 0, 0, 0',
	X =  -12.965  mm,	Y =   -548.864  mm,	Z =   -263.091  mm,
	W =  90.000 deg,	P =   0.000 deg,	R =   90.000 deg
};
P[1133]{
   GP1:
	UF : 0, UT : 6,		CONFIG : 'N U T, 0, 0, 0',
	X =  -12.188  mm,	Y =   -550.203  mm,	Z =   -263.102  mm,
	W =  90.000 deg,	P =   0.000 deg,	R =   90.000 deg
};
P[1134]{
   GP1:
	UF : 0, UT : 6,		CONFIG : 'N U T, 0, 0, 0',
	X =  -11.153  mm,	Y =   -552.031  mm,	Z =   -263.054  mm,
	W =  90.000 deg,	P =   0.000 deg,	R =   90.000 deg
};
P[1135]{
   GP1:
	UF : 0, UT : 6,		CONFIG : 'N U T, 0, 0, 0',
	X =  -9.347  mm,	Y =   -555.327  mm,	Z =   -262.816  mm,
	W =  90.000 deg,	P =   0.000 deg,	R =   90.000 deg
};
P[1136]{
   GP1:
	UF : 0, UT : 6,		CONFIG : 'N U T, 0, 0, 0',
	X =  -8.297  mm,	Y =   -557.095  mm,	Z =   -262.889  mm,
	W =  90.000 deg,	P =   0.000 deg,	R =   90.000 deg
};
P[1137]{
   GP1:
	UF : 0, UT : 6,		CONFIG : 'N U T, 0, 0, 0',
	X =  -7.300  mm,	Y =   -558.661  mm,	Z =   -263.115  mm,
	W =  90.000 deg,	P =   0.000 deg,	R =   90.000 deg
};
P[1138]{
   GP1:
	UF : 0, UT : 6,		CONFIG : 'N U T, 0, 0, 0',
	X =  -5.918  mm,	Y =   -561.069  mm,	Z =   -263.095  mm,
	W =  90.000 deg,	P =   0.000 deg,	R =   90.000 deg
};
P[1139]{
   GP1:
	UF : 0, UT : 6,		CONFIG : 'N U T, 0, 0, 0',
	X =  -5.531  mm,	Y =   -561.837  mm,	Z =   -262.958  mm,
	W =  90.000 deg,	P =   0.000 deg,	R =   90.000 deg
};
P[1140]{
   GP1:
	UF : 0, UT : 6,		CONFIG : 'N U T, 0, 0, 0',
	X =  -5.072  mm,	Y =   -562.758  mm,	Z =   -262.779  mm,
	W =  90.000 deg,	P =   0.000 deg,	R =   90.000 deg
};
P[1141]{
   GP1:
	UF : 0, UT : 6,		CONFIG : 'N U T, 0, 0, 0',
	X =  -4.608  mm,	Y =   -563.514  mm,	Z =   -262.847  mm,
	W =  90.000 deg,	P =   0.000 deg,	R =   90.000 deg
};
P[1142]{
   GP1:
	UF : 0, UT : 6,		CONFIG : 'N U T, 0, 0, 0',
	X =  -3.986  mm,	Y =   -564.449  mm,	Z =   -263.045  mm,
	W =  90.000 deg,	P =   0.000 deg,	R =   90.000 deg
};
P[1143]{
   GP1:
	UF : 0, UT : 6,		CONFIG : 'N U T, 0, 0, 0',
	X =  -3.637  mm,	Y =   -565.169  mm,	Z =   -262.883  mm,
	W =  90.000 deg,	P =   0.000 deg,	R =   90.000 deg
};
P[1144]{
   GP1:
	UF : 0, UT : 6,		CONFIG : 'N U T, 0, 0, 0',
	X =  -2.727  mm,	Y =   -566.597  mm,	Z =   -263.093  mm,
	W =  90.000 deg,	P =   0.000 deg,	R =   90.000 deg
};
P[1145]{
   GP1:
	UF : 0, UT : 6,		CONFIG : 'N U T, 0, 0, 0',
	X =  -1.284  mm,	Y =   -569.191  mm,	Z =   -262.958  mm,
	W =  90.000 deg,	P =   0.000 deg,	R =   90.000 deg
};
P[1146]{
   GP1:
	UF : 0, UT : 6,		CONFIG : 'N U T, 0, 0, 0',
	X =  0.654  mm,	Y =   -572.379  mm,	Z =   -263.193  mm,
	W =  90.000 deg,	P =   0.000 deg,	R =   90.000 deg
};
P[1147]{
   GP1:
	UF : 0, UT : 6,		CONFIG : 'N U T, 0, 0, 0',
	X =  1.441  mm,	Y =   -573.835  mm,	Z =   -263.063  mm,
	W =  90.000 deg,	P =   0.000 deg,	R =   90.000 deg
};
P[1148]{
   GP1:
	UF : 0, UT : 6,		CONFIG : 'N U T, 0, 0, 0',
	X =  2.947  mm,	Y =   -576.530  mm,	Z =   -262.942  mm,
	W =  90.000 deg,	P =   0.000 deg,	R =   90.000 deg
};
P[1149]{
   GP1:
	UF : 0, UT : 6,		CONFIG : 'N U T, 0, 0, 0',
	X =  3.718  mm,	Y =   -577.784  mm,	Z =   -263.056  mm,
	W =  90.000 deg,	P =   0.000 deg,	R =   90.000 deg
};
P[1150]{
   GP1:
	UF : 0, UT : 6,		CONFIG : 'N U T, 0, 0, 0',
	X =  4.490  mm,	Y =   -579.028  mm,	Z =   -263.186  mm,
	W =  90.000 deg,	P =   0.000 deg,	R =   90.000 deg
};
P[1151]{
   GP1:
	UF : 0, UT : 6,		CONFIG : 'N U T, 0, 0, 0',
	X =  5.020  mm,	Y =   -579.941  mm,	Z =   -263.192  mm,
	W =  90.000 deg,	P =   0.000 deg,	R =   90.000 deg
};
P[1152]{
   GP1:
	UF : 0, UT : 6,		CONFIG : 'N U T, 0, 0, 0',
	X =  5.315  mm,	Y =   -580.737  mm,	Z =   -262.795  mm,
	W =  90.000 deg,	P =   0.000 deg,	R =   90.000 deg
};
P[1153]{
   GP1:
	UF : 0, UT : 6,		CONFIG : 'N U T, 0, 0, 0',
	X =  6.943  mm,	Y =   -583.300  mm,	Z =   -263.153  mm,
	W =  90.000 deg,	P =   0.000 deg,	R =   90.000 deg
};
P[1154]{
   GP1:
	UF : 0, UT : 6,		CONFIG : 'N U T, 0, 0, 0',
	X =  7.246  mm,	Y =   -583.926  mm,	Z =   -263.012  mm,
	W =  90.000 deg,	P =   0.000 deg,	R =   90.000 deg
};
P[1155]{
   GP1:
	UF : 0, UT : 6,		CONFIG : 'N U T, 0, 0, 0',
	X =  8.915  mm,	Y =   -586.714  mm,	Z =   -263.153  mm,
	W =  90.000 deg,	P =   0.000 deg,	R =   90.000 deg
};
P[1156]{
   GP1:
	UF : 0, UT : 6,		CONFIG : 'N U T, 0, 0, 0',
	X =  9.230  mm,	Y =   -587.460  mm,	Z =   -262.874  mm,
	W =  90.000 deg,	P =   0.000 deg,	R =   90.000 deg
};
P[1157]{
   GP1:
	UF : 0, UT : 6,		CONFIG : 'N U T, 0, 0, 0',
	X =  9.572  mm,	Y =   -588.057  mm,	Z =   -262.870  mm,
	W =  90.000 deg,	P =   0.000 deg,	R =   90.000 deg
};
P[1158]{
   GP1:
	UF : 0, UT : 6,		CONFIG : 'N U T, 0, 0, 0',
	X =  10.761  mm,	Y =   -590.010  mm,	Z =   -263.016  mm,
	W =  90.000 deg,	P =   0.000 deg,	R =   90.000 deg
};
P[1159]{
   GP1:
	UF : 0, UT : 6,		CONFIG : 'N U T, 0, 0, 0',
	X =  11.366  mm,	Y =   -591.063  mm,	Z =   -263.008  mm,
	W =  90.000 deg,	P =   0.000 deg,	R =   90.000 deg
};
P[1160]{
   GP1:
	UF : 0, UT : 6,		CONFIG : 'N U T, 0, 0, 0',
	X =  11.892  mm,	Y =   -591.975  mm,	Z =   -263.008  mm,
	W =  90.000 deg,	P =   0.000 deg,	R =   90.000 deg
};
P[1161]{
   GP1:
	UF : 0, UT : 6,		CONFIG : 'N U T, 0, 0, 0',
	X =  12.330  mm,	Y =   -592.703  mm,	Z =   -263.050  mm,
	W =  90.000 deg,	P =   0.000 deg,	R =   90.000 deg
};
P[1162]{
   GP1:
	UF : 0, UT : 6,		CONFIG : 'N U T, 0, 0, 0',
	X =  15.997  mm,	Y =   -599.188  mm,	Z =   -262.865  mm,
	W =  90.000 deg,	P =   0.000 deg,	R =   90.000 deg
};
P[1163]{
   GP1:
	UF : 0, UT : 6,		CONFIG : 'N U T, 0, 0, 0',
	X =  16.751  mm,	Y =   -600.415  mm,	Z =   -262.973  mm,
	W =  90.000 deg,	P =   0.000 deg,	R =   90.000 deg
};
P[1164]{
   GP1:
	UF : 0, UT : 6,		CONFIG : 'N U T, 0, 0, 0',
	X =  17.702  mm,	Y =   -602.011  mm,	Z =   -263.046  mm,
	W =  90.000 deg,	P =   0.000 deg,	R =   90.000 deg
};
P[1165]{
   GP1:
	UF : 0, UT : 6,		CONFIG : 'N U T, 0, 0, 0',
	X =  18.634  mm,	Y =   -603.520  mm,	Z =   -263.192  mm,
	W =  90.000 deg,	P =   0.000 deg,	R =   90.000 deg
};
P[1166]{
   GP1:
	UF : 0, UT : 6,		CONFIG : 'N U T, 0, 0, 0',
	X =  19.021  mm,	Y =   -604.344  mm,	Z =   -262.976  mm,
	W =  90.000 deg,	P =   0.000 deg,	R =   90.000 deg
};
P[1167]{
   GP1:
	UF : 0, UT : 6,		CONFIG : 'N U T, 0, 0, 0',
	X =  19.368  mm,	Y =   -604.942  mm,	Z =   -262.983  mm,
	W =  90.000 deg,	P =   0.000 deg,	R =   90.000 deg
};
P[1168]{
   GP1:
	UF : 0, UT : 6,		CONFIG : 'N U T, 0, 0, 0',
	X =  20.071  mm,	Y =   -606.138  mm,	Z =   -263.012  mm,
	W =  90.000 deg,	P =   0.000 deg,	R =   90.000 deg
};
P[1169]{
   GP1:
	UF : 0, UT : 6,		CONFIG : 'N U T, 0, 0, 0',
	X =  21.511  mm,	Y =   -608.683  mm,	Z =   -262.939  mm,
	W =  90.000 deg,	P =   0.000 deg,	R =   90.000 deg
};
P[1170]{
   GP1:
	UF : 0, UT : 6,		CONFIG : 'N U T, 0, 0, 0',
	X =  21.987  mm,	Y =   -609.578  mm,	Z =   -262.843  mm,
	W =  90.000 deg,	P =   0.000 deg,	R =   90.000 deg
};
P[1171]{
   GP1:
	UF : 0, UT : 6,		CONFIG : 'N U T, 0, 0, 0',
	X =  22.409  mm,	Y =   -610.311  mm,	Z =   -262.839  mm,
	W =  90.000 deg,	P =   0.000 deg,	R =   90.000 deg
};
P[1172]{
   GP1:
	UF : 0, UT : 6,		CONFIG : 'N U T, 0, 0, 0',
	X =  22.999  mm,	Y =   -611.275  mm,	Z =   -262.919  mm,
	W =  90.000 deg,	P =   0.000 deg,	R =   90.000 deg
};
P[1173]{
   GP1:
	UF : 0, UT : 6,		CONFIG : 'N U T, 0, 0, 0',
	X =  23.748  mm,	Y =   -612.589  mm,	Z =   -262.892  mm,
	W =  90.000 deg,	P =   0.000 deg,	R =   90.000 deg
};
P[1174]{
   GP1:
	UF : 0, UT : 6,		CONFIG : 'N U T, 0, 0, 0',
	X =  24.520  mm,	Y =   -613.972  mm,	Z =   -262.830  mm,
	W =  90.000 deg,	P =   0.000 deg,	R =   90.000 deg
};
P[1175]{
   GP1:
	UF : 0, UT : 6,		CONFIG : 'N U T, 0, 0, 0',
	X =  24.891  mm,	Y =   -614.630  mm,	Z =   -262.810  mm,
	W =  90.000 deg,	P =   0.000 deg,	R =   90.000 deg
};
P[1176]{
   GP1:
	UF : 0, UT : 6,		CONFIG : 'N U T, 0, 0, 0',
	X =  25.256  mm,	Y =   -615.287  mm,	Z =   -262.776  mm,
	W =  90.000 deg,	P =   0.000 deg,	R =   90.000 deg
};
P[1177]{
   GP1:
	UF : 0, UT : 6,		CONFIG : 'N U T, 0, 0, 0',
	X =  26.208  mm,	Y =   -616.861  mm,	Z =   -262.879  mm,
	W =  90.000 deg,	P =   0.000 deg,	R =   90.000 deg
};
P[1178]{
   GP1:
	UF : 0, UT : 6,		CONFIG : 'N U T, 0, 0, 0',
	X =  27.424  mm,	Y =   -618.767  mm,	Z =   -263.159  mm,
	W =  90.000 deg,	P =   0.000 deg,	R =   90.000 deg
};
P[1179]{
   GP1:
	UF : 0, UT : 6,		CONFIG : 'N U T, 0, 0, 0',
	X =  28.304  mm,	Y =   -620.482  mm,	Z =   -262.893  mm,
	W =  90.000 deg,	P =   0.000 deg,	R =   90.000 deg
};
P[1180]{
   GP1:
	UF : 0, UT : 6,		CONFIG : 'N U T, 0, 0, 0',
	X =  29.169  mm,	Y =   -621.928  mm,	Z =   -262.966  mm,
	W =  90.000 deg,	P =   0.000 deg,	R =   90.000 deg
};
P[1181]{
   GP1:
	UF : 0, UT : 6,		CONFIG : 'N U T, 0, 0, 0',
	X =  30.058  mm,	Y =   -623.394  mm,	Z =   -263.068  mm,
	W =  90.000 deg,	P =   0.000 deg,	R =   90.000 deg
};
P[1182]{
   GP1:
	UF : 0, UT : 6,		CONFIG : 'N U T, 0, 0, 0',
	X =  31.118  mm,	Y =   -625.429  mm,	Z =   -262.789  mm,
	W =  90.000 deg,	P =   0.000 deg,	R =   90.000 deg
};
P[1183]{
   GP1:
	UF : 0, UT : 6,		CONFIG : 'N U T, 0, 0, 0',
	X =  32.827  mm,	Y =   -628.376  mm,	Z =   -262.807  mm,
	W =  90.000 deg,	P =   0.000 deg,	R =   90.000 deg
};
P[1184]{
   GP1:
	UF : 0, UT : 6,		CONFIG : 'N U T, 0, 0, 0',
	X =  33.698  mm,	Y =   -629.612  mm,	Z =   -263.190  mm,
	W =  90.000 deg,	P =   0.000 deg,	R =   90.000 deg
};
P[1185]{
   GP1:
	UF : 0, UT : 6,		CONFIG : 'N U T, 0, 0, 0',
	X =  36.077  mm,	Y =   -633.938  mm,	Z =   -262.901  mm,
	W =  90.000 deg,	P =   0.000 deg,	R =   90.000 deg
};
P[1186]{
   GP1:
	UF : 0, UT : 6,		CONFIG : 'N U T, 0, 0, 0',
	X =  36.630  mm,	Y =   -634.698  mm,	Z =   -263.179  mm,
	W =  90.000 deg,	P =   0.000 deg,	R =   90.000 deg
};
P[1187]{
   GP1:
	UF : 0, UT : 6,		CONFIG : 'N U T, 0, 0, 0',
	X =  37.787  mm,	Y =   -636.709  mm,	Z =   -263.170  mm,
	W =  90.000 deg,	P =   0.000 deg,	R =   90.000 deg
};
P[1188]{
   GP1:
	UF : 0, UT : 6,		CONFIG : 'N U T, 0, 0, 0',
	X =  38.370  mm,	Y =   -637.700  mm,	Z =   -263.196  mm,
	W =  90.000 deg,	P =   0.000 deg,	R =   90.000 deg
};
P[1189]{
   GP1:
	UF : 0, UT : 6,		CONFIG : 'N U T, 0, 0, 0',
	X =  38.847  mm,	Y =   -638.662  mm,	Z =   -263.005  mm,
	W =  90.000 deg,	P =   0.000 deg,	R =   90.000 deg
};
P[1190]{
   GP1:
	UF : 0, UT : 6,		CONFIG : 'N U T, 0, 0, 0',
	X =  40.377  mm,	Y =   -641.196  mm,	Z =   -263.169  mm,
	W =  90.000 deg,	P =   0.000 deg,	R =   90.000 deg
};
P[1191]{
   GP1:
	UF : 0, UT : 6,		CONFIG : 'N U T, 0, 0, 0',
	X =  40.859  mm,	Y =   -642.020  mm,	Z =   -263.181  mm,
	W =  90.000 deg,	P =   0.000 deg,	R =   90.000 deg
};
P[1192]{
   GP1:
	UF : 0, UT : 6,		CONFIG : 'N U T, 0, 0, 0',
	X =  42.557  mm,	Y =   -644.913  mm,	Z =   -263.248  mm,
	W =  90.000 deg,	P =   0.000 deg,	R =   90.000 deg
};
P[1193]{
   GP1:
	UF : 0, UT : 6,		CONFIG : 'N U T, 0, 0, 0',
	X =  42.859  mm,	Y =   -645.569  mm,	Z =   -263.060  mm,
	W =  90.000 deg,	P =   0.000 deg,	R =   90.000 deg
};
P[1194]{
   GP1:
	UF : 0, UT : 6,		CONFIG : 'N U T, 0, 0, 0',
	X =  44.538  mm,	Y =   -648.489  mm,	Z =   -263.044  mm,
	W =  90.000 deg,	P =   0.000 deg,	R =   90.000 deg
};
P[1195]{
   GP1:
	UF : 0, UT : 6,		CONFIG : 'N U T, 0, 0, 0',
	X =  45.041  mm,	Y =   -649.566  mm,	Z =   -262.758  mm,
	W =  90.000 deg,	P =   0.000 deg,	R =   90.000 deg
};
P[1196]{
   GP1:
	UF : 0, UT : 6,		CONFIG : 'N U T, 0, 0, 0',
	X =  47.655  mm,	Y =   -653.828  mm,	Z =   -263.129  mm,
	W =  90.000 deg,	P =   0.000 deg,	R =   90.000 deg
};
P[1197]{
   GP1:
	UF : 0, UT : 6,		CONFIG : 'N U T, 0, 0, 0',
	X =  47.992  mm,	Y =   -654.638  mm,	Z =   -262.812  mm,
	W =  90.000 deg,	P =   0.000 deg,	R =   90.000 deg
};
P[1198]{
   GP1:
	UF : 0, UT : 6,		CONFIG : 'N U T, 0, 0, 0',
	X =  48.516  mm,	Y =   -655.330  mm,	Z =   -263.114  mm,
	W =  90.000 deg,	P =   0.000 deg,	R =   90.000 deg
};
P[1199]{
   GP1:
	UF : 0, UT : 6,		CONFIG : 'N U T, 0, 0, 0',
	X =  50.670  mm,	Y =   -658.975  mm,	Z =   -263.235  mm,
	W =  90.000 deg,	P =   0.000 deg,	R =   90.000 deg
};
P[1200]{
   GP1:
	UF : 0, UT : 6,		CONFIG : 'N U T, 0, 0, 0',
	X =  52.981  mm,	Y =   -662.829  mm,	Z =   -262.791  mm,
	W =  90.000 deg,	P =   0.000 deg,	R =   90.000 deg
};
P[1201]{
   GP1:
	UF : 0, UT : 6,		CONFIG : 'N U T, 0, 0, 0',
	X =  55.056  mm,	Y =   -664.763  mm,	Z =   -263.051  mm,
	W =  90.000 deg,	P =   0.000 deg,	R =   90.000 deg
};
P[1202]{
   GP1:
	UF : 0, UT : 6,		CONFIG : 'N U T, 0, 0, 0',
	X =  56.424  mm,	Y =   -665.936  mm,	Z =   -262.777  mm,
	W =  90.000 deg,	P =   0.000 deg,	R =   90.000 deg
};
P[1203]{
   GP1:
	UF : 0, UT : 6,		CONFIG : 'N U T, 0, 0, 0',
	X =  58.211  mm,	Y =   -666.645  mm,	Z =   -263.228  mm,
	W =  90.000 deg,	P =   0.000 deg,	R =   90.000 deg
};
P[1204]{
   GP1:
	UF : 0, UT : 6,		CONFIG : 'N U T, 0, 0, 0',
	X =  61.506  mm,	Y =   -667.778  mm,	Z =   -262.853  mm,
	W =  90.000 deg,	P =   0.000 deg,	R =   90.000 deg
};
P[1205]{
   GP1:
	UF : 0, UT : 6,		CONFIG : 'N U T, 0, 0, 0',
	X =  64.902  mm,	Y =   -667.692  mm,	Z =   -263.175  mm,
	W =  90.000 deg,	P =   0.000 deg,	R =   90.000 deg
};
P[1206]{
   GP1:
	UF : 0, UT : 6,		CONFIG : 'N U T, 0, 0, 0',
	X =  67.498  mm,	Y =   -667.177  mm,	Z =   -263.089  mm,
	W =  90.000 deg,	P =   0.000 deg,	R =   90.000 deg
};
P[1207]{
   GP1:
	UF : 0, UT : 6,		CONFIG : 'N U T, 0, 0, 0',
	X =  68.598  mm,	Y =   -666.701  mm,	Z =   -263.206  mm,
	W =  90.000 deg,	P =   0.000 deg,	R =   90.000 deg
};
P[1208]{
   GP1:
	UF : 0, UT : 6,		CONFIG : 'N U T, 0, 0, 0',
	X =  72.828  mm,	Y =   -664.680  mm,	Z =   -262.792  mm,
	W =  90.000 deg,	P =   0.000 deg,	R =   90.000 deg
};
P[1209]{
   GP1:
	UF : 0, UT : 6,		CONFIG : 'N U T, 0, 0, 0',
	X =  74.459  mm,	Y =   -663.583  mm,	Z =   -263.167  mm,
	W =  90.000 deg,	P =   0.000 deg,	R =   90.000 deg
};
P[1210]{
   GP1:
	UF : 0, UT : 6,		CONFIG : 'N U T, 0, 0, 0',
	X =  75.293  mm,	Y =   -663.132  mm,	Z =   -263.095  mm,
	W =  90.000 deg,	P =   0.000 deg,	R =   90.000 deg
};
P[1211]{
   GP1:
	UF : 0, UT : 6,		CONFIG : 'N U T, 0, 0, 0',
	X =  78.529  mm,	Y =   -661.255  mm,	Z =   -263.116  mm,
	W =  90.000 deg,	P =   0.000 deg,	R =   90.000 deg
};
P[1212]{
   GP1:
	UF : 0, UT : 6,		CONFIG : 'N U T, 0, 0, 0',
	X =  82.009  mm,	Y =   -659.231  mm,	Z =   -263.150  mm,
	W =  90.000 deg,	P =   0.000 deg,	R =   90.000 deg
};
P[1213]{
   GP1:
	UF : 0, UT : 6,		CONFIG : 'N U T, 0, 0, 0',
	X =  83.551  mm,	Y =   -658.431  mm,	Z =   -262.933  mm,
	W =  90.000 deg,	P =   0.000 deg,	R =   90.000 deg
};
P[1214]{
   GP1:
	UF : 0, UT : 6,		CONFIG : 'N U T, 0, 0, 0',
	X =  84.566  mm,	Y =   -657.788  mm,	Z =   -263.069  mm,
	W =  90.000 deg,	P =   0.000 deg,	R =   90.000 deg
};
P[1215]{
   GP1:
	UF : 0, UT : 6,		CONFIG : 'N U T, 0, 0, 0',
	X =  85.714  mm,	Y =   -657.146  mm,	Z =   -263.019  mm,
	W =  90.000 deg,	P =   0.000 deg,	R =   90.000 deg
};
P[1216]{
   GP1:
	UF : 0, UT : 6,		CONFIG : 'N U T, 0, 0, 0',
	X =  86.313  mm,	Y =   -656.767  mm,	Z =   -263.098  mm,
	W =  90.000 deg,	P =   0.000 deg,	R =   90.000 deg
};
P[1217]{
   GP1:
	UF : 0, UT : 6,		CONFIG : 'N U T, 0, 0, 0',
	X =  87.438  mm,	Y =   -656.181  mm,	Z =   -262.946  mm,
	W =  90.000 deg,	P =   0.000 deg,	R =   90.000 deg
};
P[1218]{
   GP1:
	UF : 0, UT : 6,		CONFIG : 'N U T, 0, 0, 0',
	X =  90.268  mm,	Y =   -654.445  mm,	Z =   -263.191  mm,
	W =  90.000 deg,	P =   0.000 deg,	R =   90.000 deg
};
P[1219]{
   GP1:
	UF : 0, UT : 6,		CONFIG : 'N U T, 0, 0, 0',
	X =  91.260  mm,	Y =   -654.013  mm,	Z =   -262.850  mm,
	W =  90.000 deg,	P =   0.000 deg,	R =   90.000 deg
};
P[1220]{
   GP1:
	UF : 0, UT : 6,		CONFIG : 'N U T, 0, 0, 0',
	X =  96.444  mm,	Y =   -650.955  mm,	Z =   -263.010  mm,
	W =  90.000 deg,	P =   0.000 deg,	R =   90.000 deg
};
P[1221]{
   GP1:
	UF : 0, UT : 6,		CONFIG : 'N U T, 0, 0, 0',
	X =  97.162  mm,	Y =   -650.463  mm,	Z =   -263.197  mm,
	W =  90.000 deg,	P =   0.000 deg,	R =   90.000 deg
};
P[1222]{
   GP1:
	UF : 0, UT : 6,		CONFIG : 'N U T, 0, 0, 0',
	X =  98.825  mm,	Y =   -649.629  mm,	Z =   -262.891  mm,
	W =  90.000 deg,	P =   0.000 deg,	R =   90.000 deg
};
P[1223]{
   GP1:
	UF : 0, UT : 6,		CONFIG : 'N U T, 0, 0, 0',
	X =  103.339  mm,	Y =   -647.037  mm,	Z =   -262.856  mm,
	W =  90.000 deg,	P =   0.000 deg,	R =   90.000 deg
};
P[1224]{
   GP1:
	UF : 0, UT : 6,		CONFIG : 'N U T, 0, 0, 0',
	X =  105.188  mm,	Y =   -645.850  mm,	Z =   -263.145  mm,
	W =  90.000 deg,	P =   0.000 deg,	R =   90.000 deg
};
P[1225]{
   GP1:
	UF : 0, UT : 6,		CONFIG : 'N U T, 0, 0, 0',
	X =  106.201  mm,	Y =   -645.262  mm,	Z =   -263.151  mm,
	W =  90.000 deg,	P =   0.000 deg,	R =   90.000 deg
};
P[1226]{
   GP1:
	UF : 0, UT : 6,		CONFIG : 'N U T, 0, 0, 0',
	X =  107.454  mm,	Y =   -644.566  mm,	Z =   -263.086  mm,
	W =  90.000 deg,	P =   0.000 deg,	R =   90.000 deg
};
P[1227]{
   GP1:
	UF : 0, UT : 6,		CONFIG : 'N U T, 0, 0, 0',
	X =  110.464  mm,	Y =   -642.886  mm,	Z =   -262.945  mm,
	W =  90.000 deg,	P =   0.000 deg,	R =   90.000 deg
};
P[1228]{
   GP1:
	UF : 0, UT : 6,		CONFIG : 'N U T, 0, 0, 0',
	X =  114.928  mm,	Y =   -640.329  mm,	Z =   -262.897  mm,
	W =  90.000 deg,	P =   0.000 deg,	R =   90.000 deg
};
P[1229]{
   GP1:
	UF : 0, UT : 6,		CONFIG : 'N U T, 0, 0, 0',
	X =  117.048  mm,	Y =   -639.136  mm,	Z =   -262.820  mm,
	W =  90.000 deg,	P =   0.000 deg,	R =   90.000 deg
};
P[1230]{
   GP1:
	UF : 0, UT : 6,		CONFIG : 'N U T, 0, 0, 0',
	X =  121.132  mm,	Y =   -636.752  mm,	Z =   -262.882  mm,
	W =  90.000 deg,	P =   0.000 deg,	R =   90.000 deg
};
P[1231]{
   GP1:
	UF : 0, UT : 6,		CONFIG : 'N U T, 0, 0, 0',
	X =  121.812  mm,	Y =   -636.313  mm,	Z =   -262.996  mm,
	W =  90.000 deg,	P =   0.000 deg,	R =   90.000 deg
};
P[1232]{
   GP1:
	UF : 0, UT : 6,		CONFIG : 'N U T, 0, 0, 0',
	X =  123.511  mm,	Y =   -635.372  mm,	Z =   -262.899  mm,
	W =  90.000 deg,	P =   0.000 deg,	R =   90.000 deg
};
P[1233]{
   GP1:
	UF : 0, UT : 6,		CONFIG : 'N U T, 0, 0, 0',
	X =  125.558  mm,	Y =   -634.071  mm,	Z =   -263.188  mm,
	W =  90.000 deg,	P =   0.000 deg,	R =   90.000 deg
};
P[1234]{
   GP1:
	UF : 0, UT : 6,		CONFIG : 'N U T, 0, 0, 0',
	X =  126.510  mm,	Y =   -633.611  mm,	Z =   -262.969  mm,
	W =  90.000 deg,	P =   0.000 deg,	R =   90.000 deg
};
P[1235]{
   GP1:
	UF : 0, UT : 6,		CONFIG : 'N U T, 0, 0, 0',
	X =  127.767  mm,	Y =   -632.901  mm,	Z =   -262.933  mm,
	W =  90.000 deg,	P =   0.000 deg,	R =   90.000 deg
};
P[1236]{
   GP1:
	UF : 0, UT : 6,		CONFIG : 'N U T, 0, 0, 0',
	X =  129.098  mm,	Y =   -632.172  mm,	Z =   -262.835  mm,
	W =  90.000 deg,	P =   0.000 deg,	R =   90.000 deg
};
P[1237]{
   GP1:
	UF : 0, UT : 6,		CONFIG : 'N U T, 0, 0, 0',
	X =  130.371  mm,	Y =   -631.357  mm,	Z =   -263.029  mm,
	W =  90.000 deg,	P =   0.000 deg,	R =   90.000 deg
};
P[1238]{
   GP1:
	UF : 0, UT : 6,		CONFIG : 'N U T, 0, 0, 0',
	X =  131.918  mm,	Y =   -630.400  mm,	Z =   -263.184  mm,
	W =  90.000 deg,	P =   0.000 deg,	R =   90.000 deg
};
P[1239]{
   GP1:
	UF : 0, UT : 6,		CONFIG : 'N U T, 0, 0, 0',
	X =  132.618  mm,	Y =   -630.165  mm,	Z =   -262.773  mm,
	W =  90.000 deg,	P =   0.000 deg,	R =   90.000 deg
};
P[1240]{
   GP1:
	UF : 0, UT : 6,		CONFIG : 'N U T, 0, 0, 0',
	X =  133.761  mm,	Y =   -629.379  mm,	Z =   -263.080  mm,
	W =  90.000 deg,	P =   0.000 deg,	R =   90.000 deg
};
P[1241]{
   GP1:
	UF : 0, UT : 6,		CONFIG : 'N U T, 0, 0, 0',
	X =  134.542  mm,	Y =   -628.909  mm,	Z =   -263.128  mm,
	W =  90.000 deg,	P =   0.000 deg,	R =   90.000 deg
};
P[1242]{
   GP1:
	UF : 0, UT : 6,		CONFIG : 'N U T, 0, 0, 0',
	X =  135.346  mm,	Y =   -628.441  mm,	Z =   -263.136  mm,
	W =  90.000 deg,	P =   0.000 deg,	R =   90.000 deg
};
P[1243]{
   GP1:
	UF : 0, UT : 6,		CONFIG : 'N U T, 0, 0, 0',
	X =  136.285  mm,	Y =   -628.031  mm,	Z =   -262.815  mm,
	W =  90.000 deg,	P =   0.000 deg,	R =   90.000 deg
};
P[1244]{
   GP1:
	UF : 0, UT : 6,		CONFIG : 'N U T, 0, 0, 0',
	X =  136.809  mm,	Y =   -627.589  mm,	Z =   -263.153  mm,
	W =  90.000 deg,	P =   0.000 deg,	R =   90.000 deg
};
P[1245]{
   GP1:
	UF : 0, UT : 6,		CONFIG : 'N U T, 0, 0, 0',
	X =  139.128  mm,	Y =   -626.331  mm,	Z =   -262.956  mm,
	W =  90.000 deg,	P =   0.000 deg,	R =   90.000 deg
};
P[1246]{
   GP1:
	UF : 0, UT : 6,		CONFIG : 'N U T, 0, 0, 0',
	X =  139.868  mm,	Y =   -625.806  mm,	Z =   -263.192  mm,
	W =  90.000 deg,	P =   0.000 deg,	R =   90.000 deg
};
P[1247]{
   GP1:
	UF : 0, UT : 6,		CONFIG : 'N U T, 0, 0, 0',
	X =  142.204  mm,	Y =   -624.612  mm,	Z =   -262.818  mm,
	W =  90.000 deg,	P =   0.000 deg,	R =   90.000 deg
};
P[1248]{
   GP1:
	UF : 0, UT : 6,		CONFIG : 'N U T, 0, 0, 0',
	X =  145.550  mm,	Y =   -622.558  mm,	Z =   -263.114  mm,
	W =  90.000 deg,	P =   0.000 deg,	R =   90.000 deg
};
P[1249]{
   GP1:
	UF : 0, UT : 6,		CONFIG : 'N U T, 0, 0, 0',
	X =  148.248  mm,	Y =   -621.091  mm,	Z =   -262.894  mm,
	W =  90.000 deg,	P =   0.000 deg,	R =   90.000 deg
};
P[1250]{
   GP1:
	UF : 0, UT : 6,		CONFIG : 'N U T, 0, 0, 0',
	X =  148.901  mm,	Y =   -620.752  mm,	Z =   -262.802  mm,
	W =  90.000 deg,	P =   0.000 deg,	R =   90.000 deg
};
P[1251]{
   GP1:
	UF : 0, UT : 6,		CONFIG : 'N U T, 0, 0, 0',
	X =  151.252  mm,	Y =   -619.232  mm,	Z =   -263.194  mm,
	W =  90.000 deg,	P =   0.000 deg,	R =   90.000 deg
};
P[1252]{
   GP1:
	UF : 0, UT : 6,		CONFIG : 'N U T, 0, 0, 0',
	X =  153.038  mm,	Y =   -618.300  mm,	Z =   -262.956  mm,
	W =  90.000 deg,	P =   0.000 deg,	R =   90.000 deg
};
P[1253]{
   GP1:
	UF : 0, UT : 6,		CONFIG : 'N U T, 0, 0, 0',
	X =  154.134  mm,	Y =   -617.691  mm,	Z =   -262.897  mm,
	W =  90.000 deg,	P =   0.000 deg,	R =   90.000 deg
};
P[1254]{
   GP1:
	UF : 0, UT : 6,		CONFIG : 'N U T, 0, 0, 0',
	X =  154.855  mm,	Y =   -617.194  mm,	Z =   -263.094  mm,
	W =  90.000 deg,	P =   0.000 deg,	R =   90.000 deg
};
P[1255]{
   GP1:
	UF : 0, UT : 6,		CONFIG : 'N U T, 0, 0, 0',
	X =  158.057  mm,	Y =   -615.323  mm,	Z =   -263.145  mm,
	W =  90.000 deg,	P =   0.000 deg,	R =   90.000 deg
};
P[1256]{
   GP1:
	UF : 0, UT : 6,		CONFIG : 'N U T, 0, 0, 0',
	X =  159.000  mm,	Y =   -614.787  mm,	Z =   -263.127  mm,
	W =  90.000 deg,	P =   0.000 deg,	R =   90.000 deg
};
P[1257]{
   GP1:
	UF : 0, UT : 6,		CONFIG : 'N U T, 0, 0, 0',
	X =  160.130  mm,	Y =   -614.126  mm,	Z =   -263.147  mm,
	W =  90.000 deg,	P =   0.000 deg,	R =   90.000 deg
};
P[1258]{
   GP1:
	UF : 0, UT : 6,		CONFIG : 'N U T, 0, 0, 0',
	X =  161.095  mm,	Y =   -613.605  mm,	Z =   -263.061  mm,
	W =  90.000 deg,	P =   0.000 deg,	R =   90.000 deg
};
P[1259]{
   GP1:
	UF : 0, UT : 6,		CONFIG : 'N U T, 0, 0, 0',
	X =  162.553  mm,	Y =   -612.767  mm,	Z =   -263.052  mm,
	W =  90.000 deg,	P =   0.000 deg,	R =   90.000 deg
};
P[1260]{
   GP1:
	UF : 0, UT : 6,		CONFIG : 'N U T, 0, 0, 0',
	X =  163.698  mm,	Y =   -612.175  mm,	Z =   -262.883  mm,
	W =  90.000 deg,	P =   0.000 deg,	R =   90.000 deg
};
P[1261]{
   GP1:
	UF : 0, UT : 6,		CONFIG : 'N U T, 0, 0, 0',
	X =  164.961  mm,	Y =   -611.307  mm,	Z =   -263.219  mm,
	W =  90.000 deg,	P =   0.000 deg,	R =   90.000 deg
};
P[1262]{
   GP1:
	UF : 0, UT : 6,		CONFIG : 'N U T, 0, 0, 0',
	X =  165.911  mm,	Y =   -610.870  mm,	Z =   -262.949  mm,
	W =  90.000 deg,	P =   0.000 deg,	R =   90.000 deg
};
P[1263]{
   GP1:
	UF : 0, UT : 6,		CONFIG : 'N U T, 0, 0, 0',
	X =  166.621  mm,	Y =   -610.473  mm,	Z =   -262.918  mm,
	W =  90.000 deg,	P =   0.000 deg,	R =   90.000 deg
};
P[1264]{
   GP1:
	UF : 0, UT : 6,		CONFIG : 'N U T, 0, 0, 0',
	X =  167.843  mm,	Y =   -609.667  mm,	Z =   -263.162  mm,
	W =  90.000 deg,	P =   0.000 deg,	R =   90.000 deg
};
P[1265]{
   GP1:
	UF : 0, UT : 6,		CONFIG : 'N U T, 0, 0, 0',
	X =  170.926  mm,	Y =   -607.985  mm,	Z =   -262.924  mm,
	W =  90.000 deg,	P =   0.000 deg,	R =   90.000 deg
};
P[1266]{
   GP1:
	UF : 0, UT : 6,		CONFIG : 'N U T, 0, 0, 0',
	X =  172.162  mm,	Y =   -607.309  mm,	Z =   -262.829  mm,
	W =  90.000 deg,	P =   0.000 deg,	R =   90.000 deg
};
P[1267]{
   GP1:
	UF : 0, UT : 6,		CONFIG : 'N U T, 0, 0, 0',
	X =  173.193  mm,	Y =   -606.628  mm,	Z =   -263.038  mm,
	W =  90.000 deg,	P =   0.000 deg,	R =   90.000 deg
};
P[1268]{
   GP1:
	UF : 0, UT : 6,		CONFIG : 'N U T, 0, 0, 0',
	X =  177.791  mm,	Y =   -604.011  mm,	Z =   -262.948  mm,
	W =  90.000 deg,	P =   0.000 deg,	R =   90.000 deg
};
P[1269]{
   GP1:
	UF : 0, UT : 6,		CONFIG : 'N U T, 0, 0, 0',
	X =  178.366  mm,	Y =   -603.629  mm,	Z =   -263.070  mm,
	W =  90.000 deg,	P =   0.000 deg,	R =   90.000 deg
};
P[1270]{
   GP1:
	UF : 0, UT : 6,		CONFIG : 'N U T, 0, 0, 0',
	X =  179.338  mm,	Y =   -603.057  mm,	Z =   -263.096  mm,
	W =  90.000 deg,	P =   0.000 deg,	R =   90.000 deg
};
P[1271]{
   GP1:
	UF : 0, UT : 6,		CONFIG : 'N U T, 0, 0, 0',
	X =  181.149  mm,	Y =   -602.013  mm,	Z =   -263.091  mm,
	W =  90.000 deg,	P =   0.000 deg,	R =   90.000 deg
};
P[1272]{
   GP1:
	UF : 0, UT : 6,		CONFIG : 'N U T, 0, 0, 0',
	X =  181.768  mm,	Y =   -601.609  mm,	Z =   -263.204  mm,
	W =  90.000 deg,	P =   0.000 deg,	R =   90.000 deg
};
P[1273]{
   GP1:
	UF : 0, UT : 6,		CONFIG : 'N U T, 0, 0, 0',
	X =  185.822  mm,	Y =   -599.411  mm,	Z =   -262.859  mm,
	W =  90.000 deg,	P =   0.000 deg,	R =   90.000 deg
};
P[1274]{
   GP1:
	UF : 0, UT : 6,		CONFIG : 'N U T, 0, 0, 0',
	X =  187.271  mm,	Y =   -598.521  mm,	Z =   -262.986  mm,
	W =  90.000 deg,	P =   0.000 deg,	R =   90.000 deg
};
P[1275]{
   GP1:
	UF : 0, UT : 6,		CONFIG : 'N U T, 0, 0, 0',
	X =  188.229  mm,	Y =   -597.942  mm,	Z =   -263.050  mm,
	W =  90.000 deg,	P =   0.000 deg,	R =   90.000 deg
};
P[1276]{
   GP1:
	UF : 0, UT : 6,		CONFIG : 'N U T, 0, 0, 0',
	X =  188.874  mm,	Y =   -597.618  mm,	Z =   -262.933  mm,
	W =  90.000 deg,	P =   0.000 deg,	R =   90.000 deg
};
P[1277]{
   GP1:
	UF : 0, UT : 6,		CONFIG : 'N U T, 0, 0, 0',
	X =  189.774  mm,	Y =   -597.117  mm,	Z =   -262.889  mm,
	W =  90.000 deg,	P =   0.000 deg,	R =   90.000 deg
};
P[1278]{
   GP1:
	UF : 0, UT : 6,		CONFIG : 'N U T, 0, 0, 0',
	X =  190.268  mm,	Y =   -596.683  mm,	Z =   -263.246  mm,
	W =  90.000 deg,	P =   0.000 deg,	R =   90.000 deg
};
P[1279]{
   GP1:
	UF : 0, UT : 6,		CONFIG : 'N U T, 0, 0, 0',
	X =  191.225  mm,	Y =   -596.221  mm,	Z =   -263.027  mm,
	W =  90.000 deg,	P =   0.000 deg,	R =   90.000 deg
};
P[1280]{
   GP1:
	UF : 0, UT : 6,		CONFIG : 'N U T, 0, 0, 0',
	X =  195.531  mm,	Y =   -593.751  mm,	Z =   -262.988  mm,
	W =  90.000 deg,	P =   0.000 deg,	R =   90.000 deg
};
P[1281]{
   GP1:
	UF : 0, UT : 6,		CONFIG : 'N U T, 0, 0, 0',
	X =  197.115  mm,	Y =   -592.763  mm,	Z =   -263.168  mm,
	W =  90.000 deg,	P =   0.000 deg,	R =   90.000 deg
};
P[1282]{
   GP1:
	UF : 0, UT : 6,		CONFIG : 'N U T, 0, 0, 0',
	X =  198.204  mm,	Y =   -592.147  mm,	Z =   -263.137  mm,
	W =  90.000 deg,	P =   0.000 deg,	R =   90.000 deg
};
P[1283]{
   GP1:
	UF : 0, UT : 6,		CONFIG : 'N U T, 0, 0, 0',
	X =  198.925  mm,	Y =   -591.756  mm,	Z =   -263.073  mm,
	W =  90.000 deg,	P =   0.000 deg,	R =   90.000 deg
};
P[1284]{
   GP1:
	UF : 0, UT : 6,		CONFIG : 'N U T, 0, 0, 0',
	X =  200.279  mm,	Y =   -590.929  mm,	Z =   -263.185  mm,
	W =  90.000 deg,	P =   0.000 deg,	R =   90.000 deg
};
P[1285]{
   GP1:
	UF : 0, UT : 6,		CONFIG : 'N U T, 0, 0, 0',
	X =  201.525  mm,	Y =   -590.229  mm,	Z =   -263.139  mm,
	W =  90.000 deg,	P =   0.000 deg,	R =   90.000 deg
};
P[1286]{
   GP1:
	UF : 0, UT : 6,		CONFIG : 'N U T, 0, 0, 0',
	X =  204.282  mm,	Y =   -588.613  mm,	Z =   -263.195  mm,
	W =  90.000 deg,	P =   0.000 deg,	R =   90.000 deg
};
P[1287]{
   GP1:
	UF : 0, UT : 6,		CONFIG : 'N U T, 0, 0, 0',
	X =  210.128  mm,	Y =   -585.296  mm,	Z =   -263.054  mm,
	W =  90.000 deg,	P =   0.000 deg,	R =   90.000 deg
};
P[1288]{
   GP1:
	UF : 0, UT : 6,		CONFIG : 'N U T, 0, 0, 0',
	X =  211.317  mm,	Y =   -584.610  mm,	Z =   -263.052  mm,
	W =  90.000 deg,	P =   0.000 deg,	R =   90.000 deg
};
P[1289]{
   GP1:
	UF : 0, UT : 6,		CONFIG : 'N U T, 0, 0, 0',
	X =  214.877  mm,	Y =   -582.671  mm,	Z =   -262.770  mm,
	W =  90.000 deg,	P =   0.000 deg,	R =   90.000 deg
};
P[1290]{
   GP1:
	UF : 0, UT : 6,		CONFIG : 'N U T, 0, 0, 0',
	X =  215.882  mm,	Y =   -581.951  mm,	Z =   -263.110  mm,
	W =  90.000 deg,	P =   0.000 deg,	R =   90.000 deg
};
P[1291]{
   GP1:
	UF : 0, UT : 6,		CONFIG : 'N U T, 0, 0, 0',
	X =  217.702  mm,	Y =   -581.037  mm,	Z =   -262.776  mm,
	W =  90.000 deg,	P =   0.000 deg,	R =   90.000 deg
};
P[1292]{
   GP1:
	UF : 0, UT : 6,		CONFIG : 'N U T, 0, 0, 0',
	X =  219.218  mm,	Y =   -580.118  mm,	Z =   -262.884  mm,
	W =  90.000 deg,	P =   0.000 deg,	R =   90.000 deg
};
P[1293]{
   GP1:
	UF : 0, UT : 6,		CONFIG : 'N U T, 0, 0, 0',
	X =  220.265  mm,	Y =   -579.374  mm,	Z =   -263.222  mm,
	W =  90.000 deg,	P =   0.000 deg,	R =   90.000 deg
};
P[1294]{
   GP1:
	UF : 0, UT : 6,		CONFIG : 'N U T, 0, 0, 0',
	X =  224.280  mm,	Y =   -577.065  mm,	Z =   -263.199  mm,
	W =  90.000 deg,	P =   0.000 deg,	R =   90.000 deg
};
P[1295]{
   GP1:
	UF : 0, UT : 6,		CONFIG : 'N U T, 0, 0, 0',
	X =  225.238  mm,	Y =   -576.576  mm,	Z =   -263.045  mm,
	W =  90.000 deg,	P =   0.000 deg,	R =   90.000 deg
};
P[1296]{
   GP1:
	UF : 0, UT : 6,		CONFIG : 'N U T, 0, 0, 0',
	X =  226.137  mm,	Y =   -576.124  mm,	Z =   -262.881  mm,
	W =  90.000 deg,	P =   0.000 deg,	R =   90.000 deg
};
P[1297]{
   GP1:
	UF : 0, UT : 6,		CONFIG : 'N U T, 0, 0, 0',
	X =  227.061  mm,	Y =   -575.490  mm,	Z =   -263.124  mm,
	W =  90.000 deg,	P =   0.000 deg,	R =   90.000 deg
};
P[1298]{
   GP1:
	UF : 0, UT : 6,		CONFIG : 'N U T, 0, 0, 0',
	X =  229.997  mm,	Y =   -573.911  mm,	Z =   -262.843  mm,
	W =  90.000 deg,	P =   0.000 deg,	R =   90.000 deg
};
P[1299]{
   GP1:
	UF : 0, UT : 6,		CONFIG : 'N U T, 0, 0, 0',
	X =  230.840  mm,	Y =   -573.348  mm,	Z =   -263.028  mm,
	W =  90.000 deg,	P =   0.000 deg,	R =   90.000 deg
};
P[1300]{
   GP1:
	UF : 0, UT : 6,		CONFIG : 'N U T, 0, 0, 0',
	X =  232.212  mm,	Y =   -572.527  mm,	Z =   -263.098  mm,
	W =  90.000 deg,	P =   0.000 deg,	R =   90.000 deg
};
P[1301]{
   GP1:
	UF : 0, UT : 6,		CONFIG : 'N U T, 0, 0, 0',
	X =  233.505  mm,	Y =   -571.758  mm,	Z =   -263.150  mm,
	W =  90.000 deg,	P =   0.000 deg,	R =   90.000 deg
};
P[1302]{
   GP1:
	UF : 0, UT : 6,		CONFIG : 'N U T, 0, 0, 0',
	X =  234.370  mm,	Y =   -571.373  mm,	Z =   -262.873  mm,
	W =  90.000 deg,	P =   0.000 deg,	R =   90.000 deg
};
P[1303]{
   GP1:
	UF : 0, UT : 6,		CONFIG : 'N U T, 0, 0, 0',
	X =  236.697  mm,	Y =   -569.929  mm,	Z =   -263.119  mm,
	W =  90.000 deg,	P =   0.000 deg,	R =   90.000 deg
};
P[1304]{
   GP1:
	UF : 0, UT : 6,		CONFIG : 'N U T, 0, 0, 0',
	X =  238.052  mm,	Y =   -569.196  mm,	Z =   -263.000  mm,
	W =  90.000 deg,	P =   0.000 deg,	R =   90.000 deg
};
P[1305]{
   GP1:
	UF : 0, UT : 6,		CONFIG : 'N U T, 0, 0, 0',
	X =  239.713  mm,	Y =   -568.137  mm,	Z =   -263.242  mm,
	W =  90.000 deg,	P =   0.000 deg,	R =   90.000 deg
};
P[1306]{
   GP1:
	UF : 0, UT : 6,		CONFIG : 'N U T, 0, 0, 0',
	X =  241.437  mm,	Y =   -567.204  mm,	Z =   -263.090  mm,
	W =  90.000 deg,	P =   0.000 deg,	R =   90.000 deg
};
P[1307]{
   GP1:
	UF : 0, UT : 6,		CONFIG : 'N U T, 0, 0, 0',
	X =  242.299  mm,	Y =   -566.670  mm,	Z =   -263.178  mm,
	W =  90.000 deg,	P =   0.000 deg,	R =   90.000 deg
};
P[1308]{
   GP1:
	UF : 0, UT : 6,		CONFIG : 'N U T, 0, 0, 0',
	X =  243.163  mm,	Y =   -566.174  mm,	Z =   -263.170  mm,
	W =  90.000 deg,	P =   0.000 deg,	R =   90.000 deg
};
P[1309]{
   GP1:
	UF : 0, UT : 6,		CONFIG : 'N U T, 0, 0, 0',
	X =  243.807  mm,	Y =   -565.934  mm,	Z =   -262.850  mm,
	W =  90.000 deg,	P =   0.000 deg,	R =   90.000 deg
};
P[1310]{
   GP1:
	UF : 0, UT : 6,		CONFIG : 'N U T, 0, 0, 0',
	X =  246.504  mm,	Y =   -564.317  mm,	Z =   -262.996  mm,
	W =  90.000 deg,	P =   0.000 deg,	R =   90.000 deg
};
P[1311]{
   GP1:
	UF : 0, UT : 6,		CONFIG : 'N U T, 0, 0, 0',
	X =  247.965  mm,	Y =   -563.376  mm,	Z =   -263.232  mm,
	W =  90.000 deg,	P =   0.000 deg,	R =   90.000 deg
};
P[1312]{
   GP1:
	UF : 0, UT : 6,		CONFIG : 'N U T, 0, 0, 0',
	X =  248.950  mm,	Y =   -562.854  mm,	Z =   -263.118  mm,
	W =  90.000 deg,	P =   0.000 deg,	R =   90.000 deg
};
P[1313]{
   GP1:
	UF : 0, UT : 6,		CONFIG : 'N U T, 0, 0, 0',
	X =  250.645  mm,	Y =   -561.825  mm,	Z =   -263.241  mm,
	W =  90.000 deg,	P =   0.000 deg,	R =   90.000 deg
};
P[1314]{
   GP1:
	UF : 0, UT : 6,		CONFIG : 'N U T, 0, 0, 0',
	X =  251.759  mm,	Y =   -561.265  mm,	Z =   -263.039  mm,
	W =  90.000 deg,	P =   0.000 deg,	R =   90.000 deg
};
P[1315]{
   GP1:
	UF : 0, UT : 6,		CONFIG : 'N U T, 0, 0, 0',
	X =  253.258  mm,	Y =   -560.340  mm,	Z =   -263.183  mm,
	W =  90.000 deg,	P =   0.000 deg,	R =   90.000 deg
};
P[1316]{
   GP1:
	UF : 0, UT : 6,		CONFIG : 'N U T, 0, 0, 0',
	X =  254.102  mm,	Y =   -559.830  mm,	Z =   -263.239  mm,
	W =  90.000 deg,	P =   0.000 deg,	R =   90.000 deg
};
P[1317]{
   GP1:
	UF : 0, UT : 6,		CONFIG : 'N U T, 0, 0, 0',
	X =  255.792  mm,	Y =   -558.995  mm,	Z =   -262.898  mm,
	W =  90.000 deg,	P =   0.000 deg,	R =   90.000 deg
};
P[1318]{
   GP1:
	UF : 0, UT : 6,		CONFIG : 'N U T, 0, 0, 0',
	X =  257.450  mm,	Y =   -557.901  mm,	Z =   -263.228  mm,
	W =  90.000 deg,	P =   0.000 deg,	R =   90.000 deg
};
P[1319]{
   GP1:
	UF : 0, UT : 6,		CONFIG : 'N U T, 0, 0, 0',
	X =  258.435  mm,	Y =   -557.498  mm,	Z =   -262.826  mm,
	W =  90.000 deg,	P =   0.000 deg,	R =   90.000 deg
};
P[1320]{
   GP1:
	UF : 0, UT : 6,		CONFIG : 'N U T, 0, 0, 0',
	X =  260.817  mm,	Y =   -555.948  mm,	Z =   -263.250  mm,
	W =  90.000 deg,	P =   0.000 deg,	R =   90.000 deg
};
P[1321]{
   GP1:
	UF : 0, UT : 6,		CONFIG : 'N U T, 0, 0, 0',
	X =  261.775  mm,	Y =   -555.418  mm,	Z =   -263.195  mm,
	W =  90.000 deg,	P =   0.000 deg,	R =   90.000 deg
};
P[1322]{
   GP1:
	UF : 0, UT : 6,		CONFIG : 'N U T, 0, 0, 0',
	X =  264.172  mm,	Y =   -554.049  mm,	Z =   -263.158  mm,
	W =  90.000 deg,	P =   0.000 deg,	R =   90.000 deg
};
P[1323]{
   GP1:
	UF : 0, UT : 6,		CONFIG : 'N U T, 0, 0, 0',
	X =  267.750  mm,	Y =   -551.953  mm,	Z =   -263.231  mm,
	W =  90.000 deg,	P =   0.000 deg,	R =   90.000 deg
};
P[1324]{
   GP1:
	UF : 0, UT : 6,		CONFIG : 'N U T, 0, 0, 0',
	X =  269.249  mm,	Y =   -551.123  mm,	Z =   -263.143  mm,
	W =  90.000 deg,	P =   0.000 deg,	R =   90.000 deg
};
P[1325]{
   GP1:
	UF : 0, UT : 6,		CONFIG : 'N U T, 0, 0, 0',
	X =  270.166  mm,	Y =   -550.568  mm,	Z =   -263.207  mm,
	W =  90.000 deg,	P =   0.000 deg,	R =   90.000 deg
};
P[1326]{
   GP1:
	UF : 0, UT : 6,		CONFIG : 'N U T, 0, 0, 0',
	X =  272.700  mm,	Y =   -549.133  mm,	Z =   -263.138  mm,
	W =  90.000 deg,	P =   0.000 deg,	R =   90.000 deg
};
P[1327]{
   GP1:
	UF : 0, UT : 6,		CONFIG : 'N U T, 0, 0, 0',
	X =  275.577  mm,	Y =   -547.561  mm,	Z =   -262.922  mm,
	W =  90.000 deg,	P =   0.000 deg,	R =   90.000 deg
};
P[1328]{
   GP1:
	UF : 0, UT : 6,		CONFIG : 'N U T, 0, 0, 0',
	X =  277.655  mm,	Y =   -546.326  mm,	Z =   -263.006  mm,
	W =  90.000 deg,	P =   0.000 deg,	R =   90.000 deg
};
P[1329]{
   GP1:
	UF : 0, UT : 6,		CONFIG : 'N U T, 0, 0, 0',
	X =  278.466  mm,	Y =   -545.857  mm,	Z =   -263.009  mm,
	W =  90.000 deg,	P =   0.000 deg,	R =   90.000 deg
};
P[1330]{
   GP1:
	UF : 0, UT : 6,		CONFIG : 'N U T, 0, 0, 0',
	X =  279.279  mm,	Y =   -545.326  mm,	Z =   -263.156  mm,
	W =  90.000 deg,	P =   0.000 deg,	R =   90.000 deg
};
P[1331]{
   GP1:
	UF : 0, UT : 6,		CONFIG : 'N U T, 0, 0, 0',
	X =  279.924  mm,	Y =   -545.010  mm,	Z =   -263.023  mm,
	W =  90.000 deg,	P =   0.000 deg,	R =   90.000 deg
};
P[1332]{
   GP1:
	UF : 0, UT : 6,		CONFIG : 'N U T, 0, 0, 0',
	X =  281.431  mm,	Y =   -544.203  mm,	Z =   -262.870  mm,
	W =  90.000 deg,	P =   0.000 deg,	R =   90.000 deg
};
P[1333]{
   GP1:
	UF : 0, UT : 6,		CONFIG : 'N U T, 0, 0, 0',
	X =  282.122  mm,	Y =   -543.691  mm,	Z =   -263.144  mm,
	W =  90.000 deg,	P =   0.000 deg,	R =   90.000 deg
};
P[1334]{
   GP1:
	UF : 0, UT : 6,		CONFIG : 'N U T, 0, 0, 0',
	X =  284.994  mm,	Y =   -542.182  mm,	Z =   -262.782  mm,
	W =  90.000 deg,	P =   0.000 deg,	R =   90.000 deg
};
P[1335]{
   GP1:
	UF : 0, UT : 6,		CONFIG : 'N U T, 0, 0, 0',
	X =  286.954  mm,	Y =   -540.895  mm,	Z =   -263.156  mm,
	W =  90.000 deg,	P =   0.000 deg,	R =   90.000 deg
};
P[1336]{
   GP1:
	UF : 0, UT : 6,		CONFIG : 'N U T, 0, 0, 0',
	X =  288.333  mm,	Y =   -540.233  mm,	Z =   -262.829  mm,
	W =  90.000 deg,	P =   0.000 deg,	R =   90.000 deg
};
P[1337]{
   GP1:
	UF : 0, UT : 6,		CONFIG : 'N U T, 0, 0, 0',
	X =  289.468  mm,	Y =   -539.438  mm,	Z =   -263.171  mm,
	W =  90.000 deg,	P =   0.000 deg,	R =   90.000 deg
};
P[1338]{
   GP1:
	UF : 0, UT : 6,		CONFIG : 'N U T, 0, 0, 0',
	X =  292.572  mm,	Y =   -537.786  mm,	Z =   -262.831  mm,
	W =  90.000 deg,	P =   0.000 deg,	R =   90.000 deg
};
P[1339]{
   GP1:
	UF : 0, UT : 6,		CONFIG : 'N U T, 0, 0, 0',
	X =  293.731  mm,	Y =   -537.117  mm,	Z =   -262.827  mm,
	W =  90.000 deg,	P =   0.000 deg,	R =   90.000 deg
};
P[1340]{
   GP1:
	UF : 0, UT : 6,		CONFIG : 'N U T, 0, 0, 0',
	X =  295.262  mm,	Y =   -536.226  mm,	Z =   -262.847  mm,
	W =  90.000 deg,	P =   0.000 deg,	R =   90.000 deg
};
P[1341]{
   GP1:
	UF : 0, UT : 6,		CONFIG : 'N U T, 0, 0, 0',
	X =  298.626  mm,	Y =   -534.221  mm,	Z =   -262.997  mm,
	W =  90.000 deg,	P =   0.000 deg,	R =   90.000 deg
};
P[1342]{
   GP1:
	UF : 0, UT : 6,		CONFIG : 'N U T, 0, 0, 0',
	X =  299.454  mm,	Y =   -533.792  mm,	Z =   -262.879  mm,
	W =  90.000 deg,	P =   0.000 deg,	R =   90.000 deg
};
P[1343]{
   GP1:
	UF : 0, UT : 6,		CONFIG : 'N U T, 0, 0, 0',
	X =  300.895  mm,	Y =   -532.870  mm,	Z =   -263.098  mm,
	W =  90.000 deg,	P =   0.000 deg,	R =   90.000 deg
};
P[1344]{
   GP1:
	UF : 0, UT : 6,		CONFIG : 'N U T, 0, 0, 0',
	X =  302.003  mm,	Y =   -532.189  mm,	Z =   -263.198  mm,
	W =  90.000 deg,	P =   0.000 deg,	R =   90.000 deg
};
P[1345]{
   GP1:
	UF : 0, UT : 6,		CONFIG : 'N U T, 0, 0, 0',
	X =  303.110  mm,	Y =   -531.532  mm,	Z =   -263.241  mm,
	W =  90.000 deg,	P =   0.000 deg,	R =   90.000 deg
};
P[1346]{
   GP1:
	UF : 0, UT : 6,		CONFIG : 'N U T, 0, 0, 0',
	X =  305.009  mm,	Y =   -530.496  mm,	Z =   -263.093  mm,
	W =  90.000 deg,	P =   0.000 deg,	R =   90.000 deg
};
P[1347]{
   GP1:
	UF : 0, UT : 6,		CONFIG : 'N U T, 0, 0, 0',
	X =  307.721  mm,	Y =   -529.015  mm,	Z =   -262.889  mm,
	W =  90.000 deg,	P =   0.000 deg,	R =   90.000 deg
};
P[1348]{
   GP1:
	UF : 0, UT : 6,		CONFIG : 'N U T, 0, 0, 0',
	X =  311.720  mm,	Y =   -526.736  mm,	Z =   -262.814  mm,
	W =  90.000 deg,	P =   0.000 deg,	R =   90.000 deg
};
P[1349]{
   GP1:
	UF : 0, UT : 6,		CONFIG : 'N U T, 0, 0, 0',
	X =  312.712  mm,	Y =   -526.068  mm,	Z =   -263.048  mm,
	W =  90.000 deg,	P =   0.000 deg,	R =   90.000 deg
};
P[1350]{
   GP1:
	UF : 0, UT : 6,		CONFIG : 'N U T, 0, 0, 0',
	X =  315.447  mm,	Y =   -524.465  mm,	Z =   -263.105  mm,
	W =  90.000 deg,	P =   0.000 deg,	R =   90.000 deg
};
P[1351]{
   GP1:
	UF : 0, UT : 6,		CONFIG : 'N U T, 0, 0, 0',
	X =  316.670  mm,	Y =   -523.819  mm,	Z =   -262.960  mm,
	W =  90.000 deg,	P =   0.000 deg,	R =   90.000 deg
};
P[1352]{
   GP1:
	UF : 0, UT : 6,		CONFIG : 'N U T, 0, 0, 0',
	X =  318.943  mm,	Y =   -522.486  mm,	Z =   -263.008  mm,
	W =  90.000 deg,	P =   0.000 deg,	R =   90.000 deg
};
P[1353]{
   GP1:
	UF : 0, UT : 6,		CONFIG : 'N U T, 0, 0, 0',
	X =  320.058  mm,	Y =   -521.901  mm,	Z =   -262.867  mm,
	W =  90.000 deg,	P =   0.000 deg,	R =   90.000 deg
};
P[1354]{
   GP1:
	UF : 0, UT : 6,		CONFIG : 'N U T, 0, 0, 0',
	X =  320.967  mm,	Y =   -521.219  mm,	Z =   -263.248  mm,
	W =  90.000 deg,	P =   0.000 deg,	R =   90.000 deg
};
P[1355]{
   GP1:
	UF : 0, UT : 6,		CONFIG : 'N U T, 0, 0, 0',
	X =  325.714  mm,	Y =   -518.489  mm,	Z =   -263.221  mm,
	W =  90.000 deg,	P =   0.000 deg,	R =   90.000 deg
};
P[1356]{
   GP1:
	UF : 0, UT : 6,		CONFIG : 'N U T, 0, 0, 0',
	X =  326.888  mm,	Y =   -517.938  mm,	Z =   -262.914  mm,
	W =  90.000 deg,	P =   0.000 deg,	R =   90.000 deg
};
P[1357]{
   GP1:
	UF : 0, UT : 6,		CONFIG : 'N U T, 0, 0, 0',
	X =  327.963  mm,	Y =   -517.289  mm,	Z =   -262.982  mm,
	W =  90.000 deg,	P =   0.000 deg,	R =   90.000 deg
};
P[1358]{
   GP1:
	UF : 0, UT : 6,		CONFIG : 'N U T, 0, 0, 0',
	X =  330.463  mm,	Y =   -515.763  mm,	Z =   -263.181  mm,
	W =  90.000 deg,	P =   0.000 deg,	R =   90.000 deg
};
P[1359]{
   GP1:
	UF : 0, UT : 6,		CONFIG : 'N U T, 0, 0, 0',
	X =  332.740  mm,	Y =   -514.454  mm,	Z =   -263.168  mm,
	W =  90.000 deg,	P =   0.000 deg,	R =   90.000 deg
};
P[1360]{
   GP1:
	UF : 0, UT : 6,		CONFIG : 'N U T, 0, 0, 0',
	X =  333.973  mm,	Y =   -513.775  mm,	Z =   -263.090  mm,
	W =  90.000 deg,	P =   0.000 deg,	R =   90.000 deg
};
P[1361]{
   GP1:
	UF : 0, UT : 6,		CONFIG : 'N U T, 0, 0, 0',
	X =  334.887  mm,	Y =   -513.258  mm,	Z =   -263.061  mm,
	W =  90.000 deg,	P =   0.000 deg,	R =   90.000 deg
};
P[1362]{
   GP1:
	UF : 0, UT : 6,		CONFIG : 'N U T, 0, 0, 0',
	X =  337.236  mm,	Y =   -511.963  mm,	Z =   -262.914  mm,
	W =  90.000 deg,	P =   0.000 deg,	R =   90.000 deg
};
P[1363]{
   GP1:
	UF : 0, UT : 6,		CONFIG : 'N U T, 0, 0, 0',
	X =  339.992  mm,	Y =   -510.303  mm,	Z =   -263.080  mm,
	W =  90.000 deg,	P =   0.000 deg,	R =   90.000 deg
};
P[1364]{
   GP1:
	UF : 0, UT : 6,		CONFIG : 'N U T, 0, 0, 0',
	X =  341.052  mm,	Y =   -509.823  mm,	Z =   -262.758  mm,
	W =  90.000 deg,	P =   0.000 deg,	R =   90.000 deg
};
P[1365]{
   GP1:
	UF : 0, UT : 6,		CONFIG : 'N U T, 0, 0, 0',
	X =  345.105  mm,	Y =   -507.391  mm,	Z =   -262.980  mm,
	W =  90.000 deg,	P =   0.000 deg,	R =   90.000 deg
};
P[1366]{
   GP1:
	UF : 0, UT : 6,		CONFIG : 'N U T, 0, 0, 0',
	X =  347.854  mm,	Y =   -505.693  mm,	Z =   -263.251  mm,
	W =  90.000 deg,	P =   0.000 deg,	R =   90.000 deg
};
P[1367]{
   GP1:
	UF : 0, UT : 6,		CONFIG : 'N U T, 0, 0, 0',
	X =  350.548  mm,	Y =   -504.269  mm,	Z =   -262.932  mm,
	W =  90.000 deg,	P =   0.000 deg,	R =   90.000 deg
};
P[1368]{
   GP1:
	UF : 0, UT : 6,		CONFIG : 'N U T, 0, 0, 0',
	X =  351.403  mm,	Y =   -503.703  mm,	Z =   -263.108  mm,
	W =  90.000 deg,	P =   0.000 deg,	R =   90.000 deg
};
P[1369]{
   GP1:
	UF : 0, UT : 6,		CONFIG : 'N U T, 0, 0, 0',
	X =  352.290  mm,	Y =   -503.144  mm,	Z =   -263.221  mm,
	W =  90.000 deg,	P =   0.000 deg,	R =   90.000 deg
};
P[1370]{
   GP1:
	UF : 0, UT : 6,		CONFIG : 'N U T, 0, 0, 0',
	X =  354.617  mm,	Y =   -501.867  mm,	Z =   -263.061  mm,
	W =  90.000 deg,	P =   0.000 deg,	R =   90.000 deg
};
P[1371]{
   GP1:
	UF : 0, UT : 6,		CONFIG : 'N U T, 0, 0, 0',
	X =  355.749  mm,	Y =   -501.226  mm,	Z =   -263.030  mm,
	W =  90.000 deg,	P =   0.000 deg,	R =   90.000 deg
};
P[1372]{
   GP1:
	UF : 0, UT : 6,		CONFIG : 'N U T, 0, 0, 0',
	X =  356.644  mm,	Y =   -500.802  mm,	Z =   -262.803  mm,
	W =  90.000 deg,	P =   0.000 deg,	R =   90.000 deg
};
P[1373]{
   GP1:
	UF : 0, UT : 6,		CONFIG : 'N U T, 0, 0, 0',
	X =  357.254  mm,	Y =   -500.312  mm,	Z =   -263.140  mm,
	W =  90.000 deg,	P =   0.000 deg,	R =   90.000 deg
};
P[1374]{
   GP1:
	UF : 0, UT : 6,		CONFIG : 'N U T, 0, 0, 0',
	X =  357.923  mm,	Y =   -499.936  mm,	Z =   -263.114  mm,
	W =  90.000 deg,	P =   0.000 deg,	R =   90.000 deg
};
P[1375]{
   GP1:
	UF : 0, UT : 6,		CONFIG : 'N U T, 0, 0, 0',
	X =  361.634  mm,	Y =   -497.787  mm,	Z =   -263.129  mm,
	W =  90.000 deg,	P =   0.000 deg,	R =   90.000 deg
};
P[1376]{
   GP1:
	UF : 0, UT : 6,		CONFIG : 'N U T, 0, 0, 0',
	X =  363.394  mm,	Y =   -496.902  mm,	Z =   -262.811  mm,
	W =  90.000 deg,	P =   0.000 deg,	R =   90.000 deg
};
P[1377]{
   GP1:
	UF : 0, UT : 6,		CONFIG : 'N U T, 0, 0, 0',
	X =  366.297  mm,	Y =   -495.232  mm,	Z =   -262.796  mm,
	W =  90.000 deg,	P =   0.000 deg,	R =   90.000 deg
};
P[1378]{
   GP1:
	UF : 0, UT : 6,		CONFIG : 'N U T, 0, 0, 0',
	X =  368.664  mm,	Y =   -493.843  mm,	Z =   -262.851  mm,
	W =  90.000 deg,	P =   0.000 deg,	R =   90.000 deg
};
P[1379]{
   GP1:
	UF : 0, UT : 6,		CONFIG : 'N U T, 0, 0, 0',
	X =  370.170  mm,	Y =   -492.882  mm,	Z =   -263.072  mm,
	W =  90.000 deg,	P =   0.000 deg,	R =   90.000 deg
};
P[1380]{
   GP1:
	UF : 0, UT : 6,		CONFIG : 'N U T, 0, 0, 0',
	X =  371.468  mm,	Y =   -492.061  mm,	Z =   -263.245  mm,
	W =  90.000 deg,	P =   0.000 deg,	R =   90.000 deg
};
P[1381]{
   GP1:
	UF : 0, UT : 6,		CONFIG : 'N U T, 0, 0, 0',
	X =  372.790  mm,	Y =   -491.488  mm,	Z =   -262.784  mm,
	W =  90.000 deg,	P =   0.000 deg,	R =   90.000 deg
};
P[1382]{
   GP1:
	UF : 0, UT : 6,		CONFIG : 'N U T, 0, 0, 0',
	X =  373.679  mm,	Y =   -490.886  mm,	Z =   -262.999  mm,
	W =  90.000 deg,	P =   0.000 deg,	R =   90.000 deg
};
P[1383]{
   GP1:
	UF : 0, UT : 6,		CONFIG : 'N U T, 0, 0, 0',
	X =  376.501  mm,	Y =   -489.298  mm,	Z =   -262.898  mm,
	W =  90.000 deg,	P =   0.000 deg,	R =   90.000 deg
};
P[1384]{
   GP1:
	UF : 0, UT : 6,		CONFIG : 'N U T, 0, 0, 0',
	X =  377.056  mm,	Y =   -488.868  mm,	Z =   -263.165  mm,
	W =  90.000 deg,	P =   0.000 deg,	R =   90.000 deg
};
P[1385]{
   GP1:
	UF : 0, UT : 6,		CONFIG : 'N U T, 0, 0, 0',
	X =  377.616  mm,	Y =   -488.512  mm,	Z =   -263.240  mm,
	W =  90.000 deg,	P =   0.000 deg,	R =   90.000 deg
};
P[1386]{
   GP1:
	UF : 0, UT : 6,		CONFIG : 'N U T, 0, 0, 0',
	X =  378.282  mm,	Y =   -488.267  mm,	Z =   -262.906  mm,
	W =  90.000 deg,	P =   0.000 deg,	R =   90.000 deg
};
P[1387]{
   GP1:
	UF : 0, UT : 6,		CONFIG : 'N U T, 0, 0, 0',
	X =  379.856  mm,	Y =   -487.370  mm,	Z =   -262.874  mm,
	W =  90.000 deg,	P =   0.000 deg,	R =   90.000 deg
};
P[1388]{
   GP1:
	UF : 0, UT : 6,		CONFIG : 'N U T, 0, 0, 0',
	X =  382.883  mm,	Y =   -485.631  mm,	Z =   -262.856  mm,
	W =  90.000 deg,	P =   0.000 deg,	R =   90.000 deg
};
P[1389]{
   GP1:
	UF : 0, UT : 6,		CONFIG : 'N U T, 0, 0, 0',
	X =  385.836  mm,	Y =   -483.859  mm,	Z =   -263.016  mm,
	W =  90.000 deg,	P =   0.000 deg,	R =   90.000 deg
};
P[1390]{
   GP1:
	UF : 0, UT : 6,		CONFIG : 'N U T, 0, 0, 0',
	X =  388.653  mm,	Y =   -482.291  mm,	Z =   -262.874  mm,
	W =  90.000 deg,	P =   0.000 deg,	R =   90.000 deg
};
P[1391]{
   GP1:
	UF : 0, UT : 6,		CONFIG : 'N U T, 0, 0, 0',
	X =  392.774  mm,	Y =   -479.851  mm,	Z =   -263.023  mm,
	W =  90.000 deg,	P =   0.000 deg,	R =   90.000 deg
};
P[1392]{
   GP1:
	UF : 0, UT : 6,		CONFIG : 'N U T, 0, 0, 0',
	X =  394.154  mm,	Y =   -478.985  mm,	Z =   -263.191  mm,
	W =  90.000 deg,	P =   0.000 deg,	R =   90.000 deg
};
P[1393]{
   GP1:
	UF : 0, UT : 6,		CONFIG : 'N U T, 0, 0, 0',
	X =  394.765  mm,	Y =   -478.697  mm,	Z =   -263.035  mm,
	W =  90.000 deg,	P =   0.000 deg,	R =   90.000 deg
};
P[1394]{
   GP1:
	UF : 0, UT : 6,		CONFIG : 'N U T, 0, 0, 0',
	X =  395.353  mm,	Y =   -478.328  mm,	Z =   -263.104  mm,
	W =  90.000 deg,	P =   0.000 deg,	R =   90.000 deg
};
P[1395]{
   GP1:
	UF : 0, UT : 6,		CONFIG : 'N U T, 0, 0, 0',
	X =  396.474  mm,	Y =   -477.801  mm,	Z =   -262.812  mm,
	W =  90.000 deg,	P =   0.000 deg,	R =   90.000 deg
};
P[1396]{
   GP1:
	UF : 0, UT : 6,		CONFIG : 'N U T, 0, 0, 0',
	X =  397.451  mm,	Y =   -477.099  mm,	Z =   -263.150  mm,
	W =  90.000 deg,	P =   0.000 deg,	R =   90.000 deg
};
P[1397]{
   GP1:
	UF : 0, UT : 6,		CONFIG : 'N U T, 0, 0, 0',
	X =  398.221  mm,	Y =   -476.718  mm,	Z =   -262.992  mm,
	W =  90.000 deg,	P =   0.000 deg,	R =   90.000 deg
};
P[1398]{
   GP1:
	UF : 0, UT : 6,		CONFIG : 'N U T, 0, 0, 0',
	X =  398.794  mm,	Y =   -476.326  mm,	Z =   -263.142  mm,
	W =  90.000 deg,	P =   0.000 deg,	R =   90.000 deg
};
P[1399]{
   GP1:
	UF : 0, UT : 6,		CONFIG : 'N U T, 0, 0, 0',
	X =  399.784  mm,	Y =   -475.825  mm,	Z =   -262.969  mm,
	W =  90.000 deg,	P =   0.000 deg,	R =   90.000 deg
};
P[1400]{
   GP1:
	UF : 0, UT : 6,		CONFIG : 'N U T, 0, 0, 0',
	X =  402.283  mm,	Y =   -474.319  mm,	Z =   -263.125  mm,
	W =  90.000 deg,	P =   0.000 deg,	R =   90.000 deg
};
P[1401]{
   GP1:
	UF : 0, UT : 6,		CONFIG : 'N U T, 0, 0, 0',
	X =  403.539  mm,	Y =   -473.676  mm,	Z =   -262.922  mm,
	W =  90.000 deg,	P =   0.000 deg,	R =   90.000 deg
};
P[1402]{
   GP1:
	UF : 0, UT : 6,		CONFIG : 'N U T, 0, 0, 0',
	X =  404.937  mm,	Y =   -472.743  mm,	Z =   -263.228  mm,
	W =  90.000 deg,	P =   0.000 deg,	R =   90.000 deg
};
P[1403]{
   GP1:
	UF : 0, UT : 6,		CONFIG : 'N U T, 0, 0, 0',
	X =  405.649  mm,	Y =   -472.518  mm,	Z =   -262.780  mm,
	W =  90.000 deg,	P =   0.000 deg,	R =   90.000 deg
};
P[1404]{
   GP1:
	UF : 0, UT : 6,		CONFIG : 'N U T, 0, 0, 0',
	X =  406.516  mm,	Y =   -471.948  mm,	Z =   -262.945  mm,
	W =  90.000 deg,	P =   0.000 deg,	R =   90.000 deg
};
P[1405]{
   GP1:
	UF : 0, UT : 6,		CONFIG : 'N U T, 0, 0, 0',
	X =  407.576  mm,	Y =   -471.282  mm,	Z =   -263.077  mm,
	W =  90.000 deg,	P =   0.000 deg,	R =   90.000 deg
};
P[1406]{
   GP1:
	UF : 0, UT : 6,		CONFIG : 'N U T, 0, 0, 0',
	X =  408.347  mm,	Y =   -470.799  mm,	Z =   -263.167  mm,
	W =  90.000 deg,	P =   0.000 deg,	R =   90.000 deg
};
P[1407]{
   GP1:
	UF : 0, UT : 6,		CONFIG : 'N U T, 0, 0, 0',
	X =  409.011  mm,	Y =   -470.563  mm,	Z =   -262.812  mm,
	W =  90.000 deg,	P =   0.000 deg,	R =   90.000 deg
};
P[1408]{
   GP1:
	UF : 0, UT : 6,		CONFIG : 'N U T, 0, 0, 0',
	X =  410.400  mm,	Y =   -469.742  mm,	Z =   -262.856  mm,
	W =  90.000 deg,	P =   0.000 deg,	R =   90.000 deg
};
P[1409]{
   GP1:
	UF : 0, UT : 6,		CONFIG : 'N U T, 0, 0, 0',
	X =  412.594  mm,	Y =   -468.321  mm,	Z =   -263.231  mm,
	W =  90.000 deg,	P =   0.000 deg,	R =   90.000 deg
};
P[1410]{
   GP1:
	UF : 0, UT : 6,		CONFIG : 'N U T, 0, 0, 0',
	X =  414.946  mm,	Y =   -466.999  mm,	Z =   -263.143  mm,
	W =  90.000 deg,	P =   0.000 deg,	R =   90.000 deg
};
P[1411]{
   GP1:
	UF : 0, UT : 6,		CONFIG : 'N U T, 0, 0, 0',
	X =  416.991  mm,	Y =   -465.774  mm,	Z =   -263.251  mm,
	W =  90.000 deg,	P =   0.000 deg,	R =   90.000 deg
};
P[1412]{
   GP1:
	UF : 0, UT : 6,		CONFIG : 'N U T, 0, 0, 0',
	X =  417.770  mm,	Y =   -465.346  mm,	Z =   -263.198  mm,
	W =  90.000 deg,	P =   0.000 deg,	R =   90.000 deg
};
P[1413]{
   GP1:
	UF : 0, UT : 6,		CONFIG : 'N U T, 0, 0, 0',
	X =  418.799  mm,	Y =   -464.784  mm,	Z =   -263.122  mm,
	W =  90.000 deg,	P =   0.000 deg,	R =   90.000 deg
};
P[1414]{
   GP1:
	UF : 0, UT : 6,		CONFIG : 'N U T, 0, 0, 0',
	X =  419.998  mm,	Y =   -464.104  mm,	Z =   -263.092  mm,
	W =  90.000 deg,	P =   0.000 deg,	R =   90.000 deg
};
P[1415]{
   GP1:
	UF : 0, UT : 6,		CONFIG : 'N U T, 0, 0, 0',
	X =  422.234  mm,	Y =   -462.781  mm,	Z =   -263.167  mm,
	W =  90.000 deg,	P =   0.000 deg,	R =   90.000 deg
};
P[1416]{
   GP1:
	UF : 0, UT : 6,		CONFIG : 'N U T, 0, 0, 0',
	X =  425.163  mm,	Y =   -461.169  mm,	Z =   -262.976  mm,
	W =  90.000 deg,	P =   0.000 deg,	R =   90.000 deg
};
P[1417]{
   GP1:
	UF : 0, UT : 6,		CONFIG : 'N U T, 0, 0, 0',
	X =  425.902  mm,	Y =   -460.767  mm,	Z =   -262.916  mm,
	W =  90.000 deg,	P =   0.000 deg,	R =   90.000 deg
};
P[1418]{
   GP1:
	UF : 0, UT : 6,		CONFIG : 'N U T, 0, 0, 0',
	X =  426.977  mm,	Y =   -460.078  mm,	Z =   -263.080  mm,
	W =  90.000 deg,	P =   0.000 deg,	R =   90.000 deg
};
P[1419]{
   GP1:
	UF : 0, UT : 6,		CONFIG : 'N U T, 0, 0, 0',
	X =  430.471  mm,	Y =   -458.037  mm,	Z =   -263.139  mm,
	W =  90.000 deg,	P =   0.000 deg,	R =   90.000 deg
};
P[1420]{
   GP1:
	UF : 0, UT : 6,		CONFIG : 'N U T, 0, 0, 0',
	X =  432.288  mm,	Y =   -456.993  mm,	Z =   -263.128  mm,
	W =  90.000 deg,	P =   0.000 deg,	R =   90.000 deg
};
P[1421]{
   GP1:
	UF : 0, UT : 6,		CONFIG : 'N U T, 0, 0, 0',
	X =  433.285  mm,	Y =   -456.532  mm,	Z =   -262.848  mm,
	W =  90.000 deg,	P =   0.000 deg,	R =   90.000 deg
};
P[1422]{
   GP1:
	UF : 0, UT : 6,		CONFIG : 'N U T, 0, 0, 0',
	X =  437.182  mm,	Y =   -454.156  mm,	Z =   -263.155  mm,
	W =  90.000 deg,	P =   0.000 deg,	R =   90.000 deg
};
P[1423]{
   GP1:
	UF : 0, UT : 6,		CONFIG : 'N U T, 0, 0, 0',
	X =  437.926  mm,	Y =   -453.724  mm,	Z =   -263.159  mm,
	W =  90.000 deg,	P =   0.000 deg,	R =   90.000 deg
};
P[1424]{
   GP1:
	UF : 0, UT : 6,		CONFIG : 'N U T, 0, 0, 0',
	X =  439.269  mm,	Y =   -452.929  mm,	Z =   -263.207  mm,
	W =  90.000 deg,	P =   0.000 deg,	R =   90.000 deg
};
P[1425]{
   GP1:
	UF : 0, UT : 6,		CONFIG : 'N U T, 0, 0, 0',
	X =  441.128  mm,	Y =   -451.979  mm,	Z =   -262.908  mm,
	W =  90.000 deg,	P =   0.000 deg,	R =   90.000 deg
};
P[1426]{
   GP1:
	UF : 0, UT : 6,		CONFIG : 'N U T, 0, 0, 0',
	X =  441.912  mm,	Y =   -451.484  mm,	Z =   -263.010  mm,
	W =  90.000 deg,	P =   0.000 deg,	R =   90.000 deg
};
P[1427]{
   GP1:
	UF : 0, UT : 6,		CONFIG : 'N U T, 0, 0, 0',
	X =  442.912  mm,	Y =   -450.890  mm,	Z =   -263.050  mm,
	W =  90.000 deg,	P =   0.000 deg,	R =   90.000 deg
};
P[1428]{
   GP1:
	UF : 0, UT : 6,		CONFIG : 'N U T, 0, 0, 0',
	X =  444.376  mm,	Y =   -449.988  mm,	Z =   -263.189  mm,
	W =  90.000 deg,	P =   0.000 deg,	R =   90.000 deg
};
P[1429]{
   GP1:
	UF : 0, UT : 6,		CONFIG : 'N U T, 0, 0, 0',
	X =  446.864  mm,	Y =   -448.549  mm,	Z =   -263.194  mm,
	W =  90.000 deg,	P =   0.000 deg,	R =   90.000 deg
};
P[1430]{
   GP1:
	UF : 0, UT : 6,		CONFIG : 'N U T, 0, 0, 0',
	X =  448.066  mm,	Y =   -447.906  mm,	Z =   -263.070  mm,
	W =  90.000 deg,	P =   0.000 deg,	R =   90.000 deg
};
P[1431]{
   GP1:
	UF : 0, UT : 6,		CONFIG : 'N U T, 0, 0, 0',
	X =  449.325  mm,	Y =   -447.187  mm,	Z =   -263.053  mm,
	W =  90.000 deg,	P =   0.000 deg,	R =   90.000 deg
};
P[1432]{
   GP1:
	UF : 0, UT : 6,		CONFIG : 'N U T, 0, 0, 0',
	X =  452.277  mm,	Y =   -445.444  mm,	Z =   -263.143  mm,
	W =  90.000 deg,	P =   0.000 deg,	R =   90.000 deg
};
P[1433]{
   GP1:
	UF : 0, UT : 6,		CONFIG : 'N U T, 0, 0, 0',
	X =  453.752  mm,	Y =   -444.580  mm,	Z =   -263.173  mm,
	W =  90.000 deg,	P =   0.000 deg,	R =   90.000 deg
};
P[1434]{
   GP1:
	UF : 0, UT : 6,		CONFIG : 'N U T, 0, 0, 0',
	X =  454.647  mm,	Y =   -444.087  mm,	Z =   -263.115  mm,
	W =  90.000 deg,	P =   0.000 deg,	R =   90.000 deg
};
P[1435]{
   GP1:
	UF : 0, UT : 6,		CONFIG : 'N U T, 0, 0, 0',
	X =  455.842  mm,	Y =   -443.377  mm,	Z =   -263.165  mm,
	W =  90.000 deg,	P =   0.000 deg,	R =   90.000 deg
};
P[1436]{
   GP1:
	UF : 0, UT : 6,		CONFIG : 'N U T, 0, 0, 0',
	X =  457.545  mm,	Y =   -442.491  mm,	Z =   -262.930  mm,
	W =  90.000 deg,	P =   0.000 deg,	R =   90.000 deg
};
P[1437]{
   GP1:
	UF : 0, UT : 6,		CONFIG : 'N U T, 0, 0, 0',
	X =  459.797  mm,	Y =   -441.207  mm,	Z =   -262.891  mm,
	W =  90.000 deg,	P =   0.000 deg,	R =   90.000 deg
};
P[1438]{
   GP1:
	UF : 0, UT : 6,		CONFIG : 'N U T, 0, 0, 0',
	X =  464.959  mm,	Y =   -438.079  mm,	Z =   -263.246  mm,
	W =  90.000 deg,	P =   0.000 deg,	R =   90.000 deg
};
P[1439]{
   GP1:
	UF : 0, UT : 6,		CONFIG : 'N U T, 0, 0, 0',
	X =  465.650  mm,	Y =   -437.776  mm,	Z =   -263.015  mm,
	W =  90.000 deg,	P =   0.000 deg,	R =   90.000 deg
};
P[1440]{
   GP1:
	UF : 0, UT : 6,		CONFIG : 'N U T, 0, 0, 0',
	X =  466.629  mm,	Y =   -437.135  mm,	Z =   -263.198  mm,
	W =  90.000 deg,	P =   0.000 deg,	R =   90.000 deg
};
P[1441]{
   GP1:
	UF : 0, UT : 6,		CONFIG : 'N U T, 0, 0, 0',
	X =  469.117  mm,	Y =   -435.701  mm,	Z =   -263.191  mm,
	W =  90.000 deg,	P =   0.000 deg,	R =   90.000 deg
};
P[1442]{
   GP1:
	UF : 0, UT : 6,		CONFIG : 'N U T, 0, 0, 0',
	X =  472.624  mm,	Y =   -433.672  mm,	Z =   -263.201  mm,
	W =  90.000 deg,	P =   0.000 deg,	R =   90.000 deg
};
P[1443]{
   GP1:
	UF : 0, UT : 6,		CONFIG : 'N U T, 0, 0, 0',
	X =  474.526  mm,	Y =   -432.605  mm,	Z =   -263.127  mm,
	W =  90.000 deg,	P =   0.000 deg,	R =   90.000 deg
};
P[1444]{
   GP1:
	UF : 0, UT : 6,		CONFIG : 'N U T, 0, 0, 0',
	X =  479.797  mm,	Y =   -429.576  mm,	Z =   -263.090  mm,
	W =  90.000 deg,	P =   0.000 deg,	R =   90.000 deg
};
P[1445]{
   GP1:
	UF : 0, UT : 6,		CONFIG : 'N U T, 0, 0, 0',
	X =  480.655  mm,	Y =   -429.090  mm,	Z =   -263.070  mm,
	W =  90.000 deg,	P =   0.000 deg,	R =   90.000 deg
};
P[1446]{
   GP1:
	UF : 0, UT : 6,		CONFIG : 'N U T, 0, 0, 0',
	X =  483.734  mm,	Y =   -427.280  mm,	Z =   -263.147  mm,
	W =  90.000 deg,	P =   0.000 deg,	R =   90.000 deg
};
P[1447]{
   GP1:
	UF : 0, UT : 6,		CONFIG : 'N U T, 0, 0, 0',
	X =  484.903  mm,	Y =   -426.714  mm,	Z =   -262.883  mm,
	W =  90.000 deg,	P =   0.000 deg,	R =   90.000 deg
};
P[1448]{
   GP1:
	UF : 0, UT : 6,		CONFIG : 'N U T, 0, 0, 0',
	X =  485.506  mm,	Y =   -426.355  mm,	Z =   -262.909  mm,
	W =  90.000 deg,	P =   0.000 deg,	R =   90.000 deg
};
P[1449]{
   GP1:
	UF : 0, UT : 6,		CONFIG : 'N U T, 0, 0, 0',
	X =  487.113  mm,	Y =   -425.351  mm,	Z =   -263.095  mm,
	W =  90.000 deg,	P =   0.000 deg,	R =   90.000 deg
};
P[1450]{
   GP1:
	UF : 0, UT : 6,		CONFIG : 'N U T, 0, 0, 0',
	X =  489.070  mm,	Y =   -424.224  mm,	Z =   -263.087  mm,
	W =  90.000 deg,	P =   0.000 deg,	R =   90.000 deg
};
P[1451]{
   GP1:
	UF : 0, UT : 6,		CONFIG : 'N U T, 0, 0, 0',
	X =  491.520  mm,	Y =   -422.871  mm,	Z =   -262.938  mm,
	W =  90.000 deg,	P =   0.000 deg,	R =   90.000 deg
};
P[1452]{
   GP1:
	UF : 0, UT : 6,		CONFIG : 'N U T, 0, 0, 0',
	X =  492.065  mm,	Y =   -422.430  mm,	Z =   -263.242  mm,
	W =  90.000 deg,	P =   0.000 deg,	R =   90.000 deg
};
P[1453]{
   GP1:
	UF : 0, UT : 6,		CONFIG : 'N U T, 0, 0, 0',
	X =  492.930  mm,	Y =   -421.963  mm,	Z =   -263.164  mm,
	W =  90.000 deg,	P =   0.000 deg,	R =   90.000 deg
};
P[1454]{
   GP1:
	UF : 0, UT : 6,		CONFIG : 'N U T, 0, 0, 0',
	X =  493.953  mm,	Y =   -421.458  mm,	Z =   -262.956  mm,
	W =  90.000 deg,	P =   0.000 deg,	R =   90.000 deg
};
P[1455]{
   GP1:
	UF : 0, UT : 6,		CONFIG : 'N U T, 0, 0, 0',
	X =  494.833  mm,	Y =   -420.898  mm,	Z =   -263.082  mm,
	W =  90.000 deg,	P =   0.000 deg,	R =   90.000 deg
};
P[1456]{
   GP1:
	UF : 0, UT : 6,		CONFIG : 'N U T, 0, 0, 0',
	X =  495.972  mm,	Y =   -420.251  mm,	Z =   -263.056  mm,
	W =  90.000 deg,	P =   0.000 deg,	R =   90.000 deg
};
P[1457]{
   GP1:
	UF : 0, UT : 6,		CONFIG : 'N U T, 0, 0, 0',
	X =  496.524  mm,	Y =   -419.854  mm,	Z =   -263.248  mm,
	W =  90.000 deg,	P =   0.000 deg,	R =   90.000 deg
};
P[1458]{
   GP1:
	UF : 0, UT : 6,		CONFIG : 'N U T, 0, 0, 0',
	X =  498.316  mm,	Y =   -419.014  mm,	Z =   -262.775  mm,
	W =  90.000 deg,	P =   0.000 deg,	R =   90.000 deg
};
P[1459]{
   GP1:
	UF : 0, UT : 6,		CONFIG : 'N U T, 0, 0, 0',
	X =  498.890  mm,	Y =   -418.596  mm,	Z =   -262.985  mm,
	W =  90.000 deg,	P =   0.000 deg,	R =   90.000 deg
};
P[1460]{
   GP1:
	UF : 0, UT : 6,		CONFIG : 'N U T, 0, 0, 0',
	X =  500.297  mm,	Y =   -417.713  mm,	Z =   -263.158  mm,
	W =  90.000 deg,	P =   0.000 deg,	R =   90.000 deg
};
P[1461]{
   GP1:
	UF : 0, UT : 6,		CONFIG : 'N U T, 0, 0, 0',
	X =  501.964  mm,	Y =   -416.831  mm,	Z =   -262.963  mm,
	W =  90.000 deg,	P =   0.000 deg,	R =   90.000 deg
};
P[1462]{
   GP1:
	UF : 0, UT : 6,		CONFIG : 'N U T, 0, 0, 0',
	X =  503.511  mm,	Y =   -415.982  mm,	Z =   -262.852  mm,
	W =  90.000 deg,	P =   0.000 deg,	R =   90.000 deg
};
P[1463]{
   GP1:
	UF : 0, UT : 6,		CONFIG : 'N U T, 0, 0, 0',
	X =  504.903  mm,	Y =   -415.169  mm,	Z =   -262.878  mm,
	W =  90.000 deg,	P =   0.000 deg,	R =   90.000 deg
};
P[1464]{
   GP1:
	UF : 0, UT : 6,		CONFIG : 'N U T, 0, 0, 0',
	X =  505.487  mm,	Y =   -414.708  mm,	Z =   -263.176  mm,
	W =  90.000 deg,	P =   0.000 deg,	R =   90.000 deg
};
P[1465]{
   GP1:
	UF : 0, UT : 6,		CONFIG : 'N U T, 0, 0, 0',
	X =  507.425  mm,	Y =   -413.719  mm,	Z =   -262.861  mm,
	W =  90.000 deg,	P =   0.000 deg,	R =   90.000 deg
};
P[1466]{
   GP1:
	UF : 0, UT : 6,		CONFIG : 'N U T, 0, 0, 0',
	X =  509.068  mm,	Y =   -412.644  mm,	Z =   -263.168  mm,
	W =  90.000 deg,	P =   0.000 deg,	R =   90.000 deg
};
P[1467]{
   GP1:
	UF : 0, UT : 6,		CONFIG : 'N U T, 0, 0, 0',
	X =  509.894  mm,	Y =   -412.302  mm,	Z =   -262.839  mm,
	W =  90.000 deg,	P =   0.000 deg,	R =   90.000 deg
};
P[1468]{
   GP1:
	UF : 0, UT : 6,		CONFIG : 'N U T, 0, 0, 0',
	X =  510.465  mm,	Y =   -411.833  mm,	Z =   -263.178  mm,
	W =  90.000 deg,	P =   0.000 deg,	R =   90.000 deg
};
P[1469]{
   GP1:
	UF : 0, UT : 6,		CONFIG : 'N U T, 0, 0, 0',
	X =  513.523  mm,	Y =   -410.112  mm,	Z =   -263.068  mm,
	W =  90.000 deg,	P =   0.000 deg,	R =   90.000 deg
};
P[1470]{
   GP1:
	UF : 0, UT : 6,		CONFIG : 'N U T, 0, 0, 0',
	X =  514.928  mm,	Y =   -409.282  mm,	Z =   -263.115  mm,
	W =  90.000 deg,	P =   0.000 deg,	R =   90.000 deg
};
P[1471]{
   GP1:
	UF : 0, UT : 6,		CONFIG : 'N U T, 0, 0, 0',
	X =  516.712  mm,	Y =   -408.247  mm,	Z =   -263.127  mm,
	W =  90.000 deg,	P =   0.000 deg,	R =   90.000 deg
};
P[1472]{
   GP1:
	UF : 0, UT : 6,		CONFIG : 'N U T, 0, 0, 0',
	X =  517.765  mm,	Y =   -407.737  mm,	Z =   -262.892  mm,
	W =  90.000 deg,	P =   0.000 deg,	R =   90.000 deg
};
P[1473]{
   GP1:
	UF : 0, UT : 6,		CONFIG : 'N U T, 0, 0, 0',
	X =  523.198  mm,	Y =   -404.602  mm,	Z =   -262.885  mm,
	W =  90.000 deg,	P =   0.000 deg,	R =   90.000 deg
};
P[1474]{
   GP1:
	UF : 0, UT : 6,		CONFIG : 'N U T, 0, 0, 0',
	X =  526.641  mm,	Y =   -402.551  mm,	Z =   -263.041  mm,
	W =  90.000 deg,	P =   0.000 deg,	R =   90.000 deg
};
P[1475]{
   GP1:
	UF : 0, UT : 6,		CONFIG : 'N U T, 0, 0, 0',
	X =  528.759  mm,	Y =   -401.283  mm,	Z =   -263.145  mm,
	W =  90.000 deg,	P =   0.000 deg,	R =   90.000 deg
};
P[1476]{
   GP1:
	UF : 0, UT : 6,		CONFIG : 'N U T, 0, 0, 0',
	X =  529.369  mm,	Y =   -400.895  mm,	Z =   -263.233  mm,
	W =  90.000 deg,	P =   0.000 deg,	R =   90.000 deg
};
P[1477]{
   GP1:
	UF : 0, UT : 6,		CONFIG : 'N U T, 0, 0, 0',
	X =  530.120  mm,	Y =   -400.513  mm,	Z =   -263.106  mm,
	W =  90.000 deg,	P =   0.000 deg,	R =   90.000 deg
};
P[1478]{
   GP1:
	UF : 0, UT : 6,		CONFIG : 'N U T, 0, 0, 0',
	X =  530.898  mm,	Y =   -400.068  mm,	Z =   -263.099  mm,
	W =  90.000 deg,	P =   0.000 deg,	R =   90.000 deg
};
P[1479]{
   GP1:
	UF : 0, UT : 6,		CONFIG : 'N U T, 0, 0, 0',
	X =  531.874  mm,	Y =   -399.536  mm,	Z =   -262.962  mm,
	W =  90.000 deg,	P =   0.000 deg,	R =   90.000 deg
};
P[1480]{
   GP1:
	UF : 0, UT : 6,		CONFIG : 'N U T, 0, 0, 0',
	X =  534.453  mm,	Y =   -397.453  mm,	Z =   -263.155  mm,
	W =  90.000 deg,	P =   0.000 deg,	R =   90.000 deg
};
P[1481]{
   GP1:
	UF : 0, UT : 6,		CONFIG : 'N U T, 0, 0, 0',
	X =  535.384  mm,	Y =   -396.591  mm,	Z =   -262.897  mm,
	W =  90.000 deg,	P =   0.000 deg,	R =   90.000 deg
};
P[1482]{
   GP1:
	UF : 0, UT : 6,		CONFIG : 'N U T, 0, 0, 0',
	X =  536.918  mm,	Y =   -394.318  mm,	Z =   -263.035  mm,
	W =  90.000 deg,	P =   0.000 deg,	R =   90.000 deg
};
P[1483]{
   GP1:
	UF : 0, UT : 6,		CONFIG : 'N U T, 0, 0, 0',
	X =  537.512  mm,	Y =   -393.345  mm,	Z =   -262.911  mm,
	W =  90.000 deg,	P =   0.000 deg,	R =   90.000 deg
};
P[1484]{
   GP1:
	UF : 0, UT : 6,		CONFIG : 'N U T, 0, 0, 0',
	X =  538.273  mm,	Y =   -390.540  mm,	Z =   -263.190  mm,
	W =  90.000 deg,	P =   0.000 deg,	R =   90.000 deg
};
P[1485]{
   GP1:
	UF : 0, UT : 6,		CONFIG : 'N U T, 0, 0, 0',
	X =  538.492  mm,	Y =   -388.936  mm,	Z =   -263.204  mm,
	W =  90.000 deg,	P =   0.000 deg,	R =   90.000 deg
};
P[1486]{
   GP1:
	UF : 0, UT : 6,		CONFIG : 'N U T, 0, 0, 0',
	X =  536.137  mm,	Y =   -379.667  mm,	Z =   -262.874  mm,
	W =  90.000 deg,	P =   0.000 deg,	R =   90.000 deg
};
P[1487]{
   GP1:
	UF : 0, UT : 6,		CONFIG : 'N U T, 0, 0, 0',
	X =  534.949  mm,	Y =   -377.824  mm,	Z =   -263.177  mm,
	W =  90.000 deg,	P =   0.000 deg,	R =   90.000 deg
};
P[1488]{
   GP1:
	UF : 0, UT : 6,		CONFIG : 'N U T, 0, 0, 0',
	X =  534.713  mm,	Y =   -377.184  mm,	Z =   -262.852  mm,
	W =  90.000 deg,	P =   0.000 deg,	R =   90.000 deg
};
P[1489]{
   GP1:
	UF : 0, UT : 6,		CONFIG : 'N U T, 0, 0, 0',
	X =  533.014  mm,	Y =   -374.467  mm,	Z =   -263.169  mm,
	W =  90.000 deg,	P =   0.000 deg,	R =   90.000 deg
};
P[1490]{
   GP1:
	UF : 0, UT : 6,		CONFIG : 'N U T, 0, 0, 0',
	X =  532.541  mm,	Y =   -373.395  mm,	Z =   -262.814  mm,
	W =  90.000 deg,	P =   0.000 deg,	R =   90.000 deg
};
P[1491]{
   GP1:
	UF : 0, UT : 6,		CONFIG : 'N U T, 0, 0, 0',
	X =  532.010  mm,	Y =   -372.748  mm,	Z =   -263.195  mm,
	W =  90.000 deg,	P =   0.000 deg,	R =   90.000 deg
};
P[1492]{
   GP1:
	UF : 0, UT : 6,		CONFIG : 'N U T, 0, 0, 0',
	X =  530.552  mm,	Y =   -370.035  mm,	Z =   -262.933  mm,
	W =  90.000 deg,	P =   0.000 deg,	R =   90.000 deg
};
P[1493]{
   GP1:
	UF : 0, UT : 6,		CONFIG : 'N U T, 0, 0, 0',
	X =  529.590  mm,	Y =   -368.551  mm,	Z =   -263.189  mm,
	W =  90.000 deg,	P =   0.000 deg,	R =   90.000 deg
};
P[1494]{
   GP1:
	UF : 0, UT : 6,		CONFIG : 'N U T, 0, 0, 0',
	X =  528.251  mm,	Y =   -366.250  mm,	Z =   -263.213  mm,
	W =  90.000 deg,	P =   0.000 deg,	R =   90.000 deg
};
P[1495]{
   GP1:
	UF : 0, UT : 6,		CONFIG : 'N U T, 0, 0, 0',
	X =  525.119  mm,	Y =   -360.575  mm,	Z =   -262.860  mm,
	W =  90.000 deg,	P =   0.000 deg,	R =   90.000 deg
};
P[1496]{
   GP1:
	UF : 0, UT : 6,		CONFIG : 'N U T, 0, 0, 0',
	X =  524.202  mm,	Y =   -359.169  mm,	Z =   -263.117  mm,
	W =  90.000 deg,	P =   0.000 deg,	R =   90.000 deg
};
P[1497]{
   GP1:
	UF : 0, UT : 6,		CONFIG : 'N U T, 0, 0, 0',
	X =  523.621  mm,	Y =   -358.170  mm,	Z =   -263.127  mm,
	W =  90.000 deg,	P =   0.000 deg,	R =   90.000 deg
};
P[1498]{
   GP1:
	UF : 0, UT : 6,		CONFIG : 'N U T, 0, 0, 0',
	X =  522.688  mm,	Y =   -356.501  mm,	Z =   -263.054  mm,
	W =  90.000 deg,	P =   0.000 deg,	R =   90.000 deg
};
P[1499]{
   GP1:
	UF : 0, UT : 6,		CONFIG : 'N U T, 0, 0, 0',
	X =  521.452  mm,	Y =   -354.306  mm,	Z =   -262.975  mm,
	W =  90.000 deg,	P =   0.000 deg,	R =   90.000 deg
};
P[1500]{
   GP1:
	UF : 0, UT : 6,		CONFIG : 'N U T, 0, 0, 0',
	X =  520.317  mm,	Y =   -352.531  mm,	Z =   -263.242  mm,
	W =  90.000 deg,	P =   0.000 deg,	R =   90.000 deg
};
P[1501]{
   GP1:
	UF : 0, UT : 6,		CONFIG : 'N U T, 0, 0, 0',
	X =  519.798  mm,	Y =   -351.435  mm,	Z =   -262.968  mm,
	W =  90.000 deg,	P =   0.000 deg,	R =   90.000 deg
};
P[1502]{
   GP1:
	UF : 0, UT : 6,		CONFIG : 'N U T, 0, 0, 0',
	X =  518.162  mm,	Y =   -348.655  mm,	Z =   -263.042  mm,
	W =  90.000 deg,	P =   0.000 deg,	R =   90.000 deg
};
P[1503]{
   GP1:
	UF : 0, UT : 6,		CONFIG : 'N U T, 0, 0, 0',
	X =  517.724  mm,	Y =   -348.038  mm,	Z =   -263.239  mm,
	W =  90.000 deg,	P =   0.000 deg,	R =   90.000 deg
};
P[1504]{
   GP1:
	UF : 0, UT : 6,		CONFIG : 'N U T, 0, 0, 0',
	X =  517.245  mm,	Y =   -347.119  mm,	Z =   -263.117  mm,
	W =  90.000 deg,	P =   0.000 deg,	R =   90.000 deg
};
P[1505]{
   GP1:
	UF : 0, UT : 6,		CONFIG : 'N U T, 0, 0, 0',
	X =  516.837  mm,	Y =   -346.359  mm,	Z =   -263.043  mm,
	W =  90.000 deg,	P =   0.000 deg,	R =   90.000 deg
};
P[1506]{
   GP1:
	UF : 0, UT : 6,		CONFIG : 'N U T, 0, 0, 0',
	X =  515.466  mm,	Y =   -344.006  mm,	Z =   -263.069  mm,
	W =  90.000 deg,	P =   0.000 deg,	R =   90.000 deg
};
P[1507]{
   GP1:
	UF : 0, UT : 6,		CONFIG : 'N U T, 0, 0, 0',
	X =  514.611  mm,	Y =   -342.409  mm,	Z =   -262.907  mm,
	W =  90.000 deg,	P =   0.000 deg,	R =   90.000 deg
};
P[1508]{
   GP1:
	UF : 0, UT : 6,		CONFIG : 'N U T, 0, 0, 0',
	X =  513.909  mm,	Y =   -341.345  mm,	Z =   -263.120  mm,
	W =  90.000 deg,	P =   0.000 deg,	R =   90.000 deg
};
P[1509]{
   GP1:
	UF : 0, UT : 6,		CONFIG : 'N U T, 0, 0, 0',
	X =  512.043  mm,	Y =   -338.154  mm,	Z =   -263.180  mm,
	W =  90.000 deg,	P =   0.000 deg,	R =   90.000 deg
};
P[1510]{
   GP1:
	UF : 0, UT : 6,		CONFIG : 'N U T, 0, 0, 0',
	X =  509.318  mm,	Y =   -333.455  mm,	Z =   -263.207  mm,
	W =  90.000 deg,	P =   0.000 deg,	R =   90.000 deg
};
P[1511]{
   GP1:
	UF : 0, UT : 6,		CONFIG : 'N U T, 0, 0, 0',
	X =  508.597  mm,	Y =   -331.953  mm,	Z =   -262.854  mm,
	W =  90.000 deg,	P =   0.000 deg,	R =   90.000 deg
};
P[1512]{
   GP1:
	UF : 0, UT : 6,		CONFIG : 'N U T, 0, 0, 0',
	X =  507.592  mm,	Y =   -330.229  mm,	Z =   -262.875  mm,
	W =  90.000 deg,	P =   0.000 deg,	R =   90.000 deg
};
P[1513]{
   GP1:
	UF : 0, UT : 6,		CONFIG : 'N U T, 0, 0, 0',
	X =  505.044  mm,	Y =   -325.952  mm,	Z =   -263.065  mm,
	W =  90.000 deg,	P =   0.000 deg,	R =   90.000 deg
};
P[1514]{
   GP1:
	UF : 0, UT : 6,		CONFIG : 'N U T, 0, 0, 0',
	X =  503.603  mm,	Y =   -323.440  mm,	Z =   -263.042  mm,
	W =  90.000 deg,	P =   0.000 deg,	R =   90.000 deg
};
P[1515]{
   GP1:
	UF : 0, UT : 6,		CONFIG : 'N U T, 0, 0, 0',
	X =  502.314  mm,	Y =   -321.225  mm,	Z =   -263.067  mm,
	W =  90.000 deg,	P =   0.000 deg,	R =   90.000 deg
};
P[1516]{
   GP1:
	UF : 0, UT : 6,		CONFIG : 'N U T, 0, 0, 0',
	X =  501.026  mm,	Y =   -319.044  mm,	Z =   -263.139  mm,
	W =  90.000 deg,	P =   0.000 deg,	R =   90.000 deg
};
P[1517]{
   GP1:
	UF : 0, UT : 6,		CONFIG : 'N U T, 0, 0, 0',
	X =  497.746  mm,	Y =   -313.427  mm,	Z =   -263.228  mm,
	W =  90.000 deg,	P =   0.000 deg,	R =   90.000 deg
};
P[1518]{
   GP1:
	UF : 0, UT : 6,		CONFIG : 'N U T, 0, 0, 0',
	X =  496.705  mm,	Y =   -311.539  mm,	Z =   -263.106  mm,
	W =  90.000 deg,	P =   0.000 deg,	R =   90.000 deg
};
P[1519]{
   GP1:
	UF : 0, UT : 6,		CONFIG : 'N U T, 0, 0, 0',
	X =  496.114  mm,	Y =   -310.390  mm,	Z =   -262.933  mm,
	W =  90.000 deg,	P =   0.000 deg,	R =   90.000 deg
};
P[1520]{
   GP1:
	UF : 0, UT : 6,		CONFIG : 'N U T, 0, 0, 0',
	X =  495.454  mm,	Y =   -309.453  mm,	Z =   -263.220  mm,
	W =  90.000 deg,	P =   0.000 deg,	R =   90.000 deg
};
P[1521]{
   GP1:
	UF : 0, UT : 6,		CONFIG : 'N U T, 0, 0, 0',
	X =  494.864  mm,	Y =   -308.185  mm,	Z =   -262.875  mm,
	W =  90.000 deg,	P =   0.000 deg,	R =   90.000 deg
};
P[1522]{
   GP1:
	UF : 0, UT : 6,		CONFIG : 'N U T, 0, 0, 0',
	X =  493.938  mm,	Y =   -306.835  mm,	Z =   -263.232  mm,
	W =  90.000 deg,	P =   0.000 deg,	R =   90.000 deg
};
P[1523]{
   GP1:
	UF : 0, UT : 6,		CONFIG : 'N U T, 0, 0, 0',
	X =  493.393  mm,	Y =   -305.791  mm,	Z =   -263.090  mm,
	W =  90.000 deg,	P =   0.000 deg,	R =   90.000 deg
};
P[1524]{
   GP1:
	UF : 0, UT : 6,		CONFIG : 'N U T, 0, 0, 0',
	X =  492.695  mm,	Y =   -304.621  mm,	Z =   -263.143  mm,
	W =  90.000 deg,	P =   0.000 deg,	R =   90.000 deg
};
P[1525]{
   GP1:
	UF : 0, UT : 6,		CONFIG : 'N U T, 0, 0, 0',
	X =  491.913  mm,	Y =   -303.020  mm,	Z =   -262.798  mm,
	W =  90.000 deg,	P =   0.000 deg,	R =   90.000 deg
};
P[1526]{
   GP1:
	UF : 0, UT : 6,		CONFIG : 'N U T, 0, 0, 0',
	X =  491.245  mm,	Y =   -301.964  mm,	Z =   -262.941  mm,
	W =  90.000 deg,	P =   0.000 deg,	R =   90.000 deg
};
P[1527]{
   GP1:
	UF : 0, UT : 6,		CONFIG : 'N U T, 0, 0, 0',
	X =  490.810  mm,	Y =   -301.340  mm,	Z =   -263.122  mm,
	W =  90.000 deg,	P =   0.000 deg,	R =   90.000 deg
};
P[1528]{
   GP1:
	UF : 0, UT : 6,		CONFIG : 'N U T, 0, 0, 0',
	X =  489.797  mm,	Y =   -299.589  mm,	Z =   -263.128  mm,
